   1:  PR[91,3] = PR[90,3] + 56.600;
   1:L PR[91] R[100]mm/sec CNT100;
   1:  PR[91,1] = PR[90,1] + 23.637;
   1:  PR[91,2] = PR[90,2] + -23.851;
   1:  PR[91,3] = PR[90,3] + 56.612;
   1:L PR[91] R[100]mm/sec CNT100;
   1:  PR[91,1] = PR[90,1] + 29.260;
   1:  PR[91,2] = PR[90,2] + -22.769;
   1:  PR[91,3] = PR[90,3] + 56.618;
   1:L PR[91] R[100]mm/sec CNT100;
   1:  PR[91,1] = PR[90,1] + 29.704;
   1:  PR[91,2] = PR[90,2] + -22.625;
   1:  PR[91,3] = PR[90,3] + 56.637;
   1:L PR[91] R[100]mm/sec CNT100;
   1:  PR[91,1] = PR[90,1] + 30.561;
   1:  PR[91,2] = PR[90,2] + -22.294;
   1:  PR[91,3] = PR[90,3] + 56.639;
   1:L PR[91] R[100]mm/sec CNT100;
   1:  PR[91,1] = PR[90,1] + 33.444;
   1:  PR[91,2] = PR[90,2] + -20.954;
   1:  PR[91,3] = PR[90,3] + 56.642;
   1:L PR[91] R[100]mm/sec CNT100;
   1:  PR[91,1] = PR[90,1] + 37.250;
   1:  PR[91,2] = PR[90,2] + -22.447;
   1:  PR[91,3] = PR[90,3] + 56.652;
   1:L PR[91] R[100]mm/sec CNT100;
   1:  PR[91,1] = PR[90,1] + 37.514;
   1:  PR[91,2] = PR[90,2] + -22.529;
   1:  PR[91,3] = PR[90,3] + 56.666;
   1:L PR[91] R[100]mm/sec CNT100;
   1:  PR[91,1] = PR[90,1] + 38.883;
   1:  PR[91,2] = PR[90,2] + -22.892;
   1:  PR[91,3] = PR[90,3] + 56.667;
   1:L PR[91] R[100]mm/sec CNT100;
   1:  PR[91,1] = PR[90,1] + 41.909;
   1:  PR[91,2] = PR[90,2] + -23.658;
   1:  PR[91,3] = PR[90,3] + 56.671;
   1:L PR[91] R[100]mm/sec CNT100;
   1:  PR[91,1] = PR[90,1] + 45.377;
   1:  PR[91,2] = PR[90,2] + -24.220;
   1:  PR[91,3] = PR[90,3] + 56.682;
   1:L PR[91] R[100]mm/sec CNT100;
   1:  PR[91,1] = PR[90,1] + 46.524;
   1:  PR[91,2] = PR[90,2] + -24.421;
   1:  PR[91,3] = PR[90,3] + 56.693;
   1:L PR[91] R[100]mm/sec CNT100;
   1:  PR[91,1] = PR[90,1] + 50.126;
   1:  PR[91,2] = PR[90,2] + -24.627;
   1:  PR[91,3] = PR[90,3] + 56.697;
   1:L PR[91] R[100]mm/sec CNT100;
   1:  PR[91,1] = PR[90,1] + 55.050;
   1:  PR[91,2] = PR[90,2] + -24.652;
   1:  PR[91,3] = PR[90,3] + 56.709;
   1:L PR[91] R[100]mm/sec CNT100;
   1:  PR[91,1] = PR[90,1] + 55.608;
   1:  PR[91,2] = PR[90,2] + -24.620;
   1:  PR[91,3] = PR[90,3] + 56.725;
   1:L PR[91] R[100]mm/sec CNT100;
   1:  PR[91,1] = PR[90,1] + 60.745;
   1:  PR[91,2] = PR[90,2] + -23.797;
   1:  PR[91,3] = PR[90,3] + 56.727;
   1:L PR[91] R[100]mm/sec CNT100;
   1:  PR[91,1] = PR[90,1] + 62.719;
   1:  PR[91,2] = PR[90,2] + -23.452;
   1:  PR[91,3] = PR[90,3] + 56.744;
   1:L PR[91] R[100]mm/sec CNT100;
   1:  PR[91,1] = PR[90,1] + 65.264;
   1:  PR[91,2] = PR[90,2] + -22.556;
   1:  PR[91,3] = PR[90,3] + 56.751;
   1:L PR[91] R[100]mm/sec CNT100;
   1:  PR[91,1] = PR[90,1] + 69.091;
   1:  PR[91,2] = PR[90,2] + -21.163;
   1:  PR[91,3] = PR[90,3] + 56.760;
   1:L PR[91] R[100]mm/sec CNT100;
   1:  PR[91,1] = PR[90,1] + 71.668;
   1:  PR[91,2] = PR[90,2] + -19.643;
   1:  PR[91,3] = PR[90,3] + 56.773;
   1:L PR[91] R[100]mm/sec CNT100;
   1:  PR[91,1] = PR[90,1] + 74.000;
   1:  PR[91,2] = PR[90,2] + -18.185;
   1:  PR[91,3] = PR[90,3] + 56.783;
   1:L PR[91] R[100]mm/sec CNT100;
   1:  PR[91,1] = PR[90,1] + 74.562;
   1:  PR[91,2] = PR[90,2] + -17.699;
   1:  PR[91,3] = PR[90,3] + 56.792;
   1:L PR[91] R[100]mm/sec CNT100;
   1:  PR[91,1] = PR[90,1] + 77.771;
   1:  PR[91,2] = PR[90,2] + -14.617;
   1:  PR[91,3] = PR[90,3] + 56.794;
   1:L PR[91] R[100]mm/sec CNT100;
   1:  PR[91,1] = PR[90,1] + 78.956;
   1:  PR[91,2] = PR[90,2] + -12.985;
   1:  PR[91,3] = PR[90,3] + 56.809;
   1:L PR[91] R[100]mm/sec CNT100;
   1:  PR[91,1] = PR[90,1] + 80.681;
   1:  PR[91,2] = PR[90,2] + -10.394;
   1:  PR[91,3] = PR[90,3] + 56.816;
   1:L PR[91] R[100]mm/sec CNT100;
   1:  PR[91,1] = PR[90,1] + 81.711;
   1:  PR[91,2] = PR[90,2] + -7.850;
   1:  PR[91,3] = PR[90,3] + 56.826;
   1:L PR[91] R[100]mm/sec CNT100;
   1:  PR[91,1] = PR[90,1] + 82.517;
   1:  PR[91,2] = PR[90,2] + -5.690;
   1:  PR[91,3] = PR[90,3] + 56.835;
   1:L PR[91] R[100]mm/sec CNT100;
   1:  PR[91,1] = PR[90,1] + 82.929;
   1:  PR[91,2] = PR[90,2] + -2.575;
   1:  PR[91,3] = PR[90,3] + 56.843;
   1:L PR[91] R[100]mm/sec CNT100;
   1:  PR[91,1] = PR[90,1] + 83.277;
   1:  PR[91,2] = PR[90,2] + -0.677;
   1:  PR[91,3] = PR[90,3] + 56.853;
   1:L PR[91] R[100]mm/sec CNT100;
   1:  PR[91,1] = PR[90,1] + 83.183;
   1:  PR[91,2] = PR[90,2] + 0.041;
   1:  PR[91,3] = PR[90,3] + 56.859;
   1:L PR[91] R[100]mm/sec CNT100;
   1:  PR[91,1] = PR[90,1] + 82.753;
   1:  PR[91,2] = PR[90,2] + 2.220;
   1:  PR[91,3] = PR[90,3] + 56.862;
   1:L PR[91] R[100]mm/sec CNT100;
   1:  PR[91,1] = PR[90,1] + 82.512;
   1:  PR[91,2] = PR[90,2] + 4.246;
   1:  PR[91,3] = PR[90,3] + 56.869;
   1:L PR[91] R[100]mm/sec CNT100;
   1:  PR[91,1] = PR[90,1] + 81.707;
   1:  PR[91,2] = PR[90,2] + 6.399;
   1:  PR[91,3] = PR[90,3] + 56.876;
   1:L PR[91] R[100]mm/sec CNT100;
   1:  PR[91,1] = PR[90,1] + 80.678;
   1:  PR[91,2] = PR[90,2] + 8.942;
   1:  PR[91,3] = PR[90,3] + 56.883;
   1:L PR[91] R[100]mm/sec CNT100;
   1:  PR[91,1] = PR[90,1] + 78.944;
   1:  PR[91,2] = PR[90,2] + 11.541;
   1:  PR[91,3] = PR[90,3] + 56.892;
   1:L PR[91] R[100]mm/sec CNT100;
   1:  PR[91,1] = PR[90,1] + 77.761;
   1:  PR[91,2] = PR[90,2] + 13.171;
   1:  PR[91,3] = PR[90,3] + 56.903;
   1:L PR[91] R[100]mm/sec CNT100;
   1:  PR[91,1] = PR[90,1] + 74.532;
   1:  PR[91,2] = PR[90,2] + 16.264;
   1:  PR[91,3] = PR[90,3] + 56.909;
   1:L PR[91] R[100]mm/sec CNT100;
   1:  PR[91,1] = PR[90,1] + 73.976;
   1:  PR[91,2] = PR[90,2] + 16.745;
   1:  PR[91,3] = PR[90,3] + 56.924;
   1:L PR[91] R[100]mm/sec CNT100;
   1:  PR[91,1] = PR[90,1] + 71.670;
   1:  PR[91,2] = PR[90,2] + 18.183;
   1:  PR[91,3] = PR[90,3] + 56.926;
   1:L PR[91] R[100]mm/sec CNT100;
   1:  PR[91,1] = PR[90,1] + 69.055;
   1:  PR[91,2] = PR[90,2] + 19.721;
   1:  PR[91,3] = PR[90,3] + 56.935;
   1:L PR[91] R[100]mm/sec CNT100;
   1:  PR[91,1] = PR[90,1] + 65.241;
   1:  PR[91,2] = PR[90,2] + 21.101;
   1:  PR[91,3] = PR[90,3] + 56.945;
   1:L PR[91] R[100]mm/sec CNT100;
   1:  PR[91,1] = PR[90,1] + 62.707;
   1:  PR[91,2] = PR[90,2] + 21.996;
   1:  PR[91,3] = PR[90,3] + 56.959;
   1:L PR[91] R[100]mm/sec CNT100;
   1:  PR[91,1] = PR[90,1] + 60.741;
   1:  PR[91,2] = PR[90,2] + 22.335;
   1:  PR[91,3] = PR[90,3] + 56.968;
   1:L PR[91] R[100]mm/sec CNT100;
   1:  PR[91,1] = PR[90,1] + 55.634;
   1:  PR[91,2] = PR[90,2] + 23.160;
   1:  PR[91,3] = PR[90,3] + 56.974;
   1:L PR[91] R[100]mm/sec CNT100;
   1:  PR[91,1] = PR[90,1] + 55.091;
   1:  PR[91,2] = PR[90,2] + 23.191;
   1:  PR[91,3] = PR[90,3] + 56.991;
   1:L PR[91] R[100]mm/sec CNT100;
   1:  PR[91,1] = PR[90,1] + 50.139;
   1:  PR[91,2] = PR[90,2] + 23.170;
   1:  PR[91,3] = PR[90,3] + 56.993;
   1:L PR[91] R[100]mm/sec CNT100;
   1:  PR[91,1] = PR[90,1] + 46.529;
   1:  PR[91,2] = PR[90,2] + 22.962;
   1:  PR[91,3] = PR[90,3] + 57.009;
   1:L PR[91] R[100]mm/sec CNT100;
   1:  PR[91,1] = PR[90,1] + 45.377;
   1:  PR[91,2] = PR[90,2] + 22.761;
   1:  PR[91,3] = PR[90,3] + 57.021;
   1:L PR[91] R[100]mm/sec CNT100;
   1:  PR[91,1] = PR[90,1] + 41.909;
   1:  PR[91,2] = PR[90,2] + 22.199;
   1:  PR[91,3] = PR[90,3] + 57.025;
   1:L PR[91] R[100]mm/sec CNT100;
   1:  PR[91,1] = PR[90,1] + 38.883;
   1:  PR[91,2] = PR[90,2] + 21.434;
   1:  PR[91,3] = PR[90,3] + 57.037;
   1:L PR[91] R[100]mm/sec CNT100;
   1:  PR[91,1] = PR[90,1] + 37.514;
   1:  PR[91,2] = PR[90,2] + 21.070;
   1:  PR[91,3] = PR[90,3] + 57.047;
   1:L PR[91] R[100]mm/sec CNT100;
   1:  PR[91,1] = PR[90,1] + 37.250;
   1:  PR[91,2] = PR[90,2] + 20.988;
   1:  PR[91,3] = PR[90,3] + 57.052;
   1:L PR[91] R[100]mm/sec CNT100;
   1:  PR[91,1] = PR[90,1] + 33.444;
   1:  PR[91,2] = PR[90,2] + 19.495;
   1:  PR[91,3] = PR[90,3] + 57.053;
   1:L PR[91] R[100]mm/sec CNT100;
   1:  PR[91,1] = PR[90,1] + 30.562;
   1:  PR[91,2] = PR[90,2] + 20.835;
   1:  PR[91,3] = PR[90,3] + 57.066;
   1:L PR[91] R[100]mm/sec CNT100;
   1:  PR[91,1] = PR[90,1] + 29.701;
   1:  PR[91,2] = PR[90,2] + 21.168;
   1:  PR[91,3] = PR[90,3] + 57.077;
   1:L PR[91] R[100]mm/sec CNT100;
   1:  PR[91,1] = PR[90,1] + 29.320;
   1:  PR[91,2] = PR[90,2] + 21.293;
   1:  PR[91,3] = PR[90,3] + 57.080;
   1:L PR[91] R[100]mm/sec CNT100;
   1:  PR[91,1] = PR[90,1] + 25.439;
   1:  PR[91,2] = PR[90,2] + 22.057;
   1:  PR[91,3] = PR[90,3] + 57.081;
   1:L PR[91] R[100]mm/sec CNT100;
   1:  PR[91,1] = PR[90,1] + 23.646;
   1:  PR[91,2] = PR[90,2] + 22.392;
   1:  PR[91,3] = PR[90,3] + 57.094;
   1:L PR[91] R[100]mm/sec CNT100;
   1:  PR[91,1] = PR[90,1] + 21.624;
   1:  PR[91,2] = PR[90,2] + 22.312;
   1:  PR[91,3] = PR[90,3] + 57.100;
   1:L PR[91] R[100]mm/sec CNT100;
   1:  PR[91,1] = PR[90,1] + 18.051;
   1:  PR[91,2] = PR[90,2] + 22.116;
   1:  PR[91,3] = PR[90,3] + 57.107;
   1:L PR[91] R[100]mm/sec CNT100;
   1:  PR[91,1] = PR[90,1] + 15.863;
   1:  PR[91,2] = PR[90,2] + 21.519;
   1:  PR[91,3] = PR[90,3] + 57.118;
   1:L PR[91] R[100]mm/sec CNT100;
   1:  PR[91,1] = PR[90,1] + 12.714;
   1:  PR[91,2] = PR[90,2] + 20.535;
   1:  PR[91,3] = PR[90,3] + 57.126;
   1:L PR[91] R[100]mm/sec CNT100;
   1:  PR[91,1] = PR[90,1] + 10.446;
   1:  PR[91,2] = PR[90,2] + 19.306;
   1:  PR[91,3] = PR[90,3] + 57.137;
   1:L PR[91] R[100]mm/sec CNT100;
   1:  PR[91,1] = PR[90,1] + 7.875;
   1:  PR[91,2] = PR[90,2] + 17.717;
   1:  PR[91,3] = PR[90,3] + 57.145;
   1:L PR[91] R[100]mm/sec CNT100;
   1:  PR[91,1] = PR[90,1] + 6.403;
   1:  PR[91,2] = PR[90,2] + 16.502;
   1:  PR[91,3] = PR[90,3] + 57.155;
   1:L PR[91] R[100]mm/sec CNT100;
   1:  PR[91,1] = PR[90,1] + 4.585;
   1:  PR[91,2] = PR[90,2] + 14.804;
   1:  PR[91,3] = PR[90,3] + 57.162;
   1:L PR[91] R[100]mm/sec CNT100;
   1:  PR[91,1] = PR[90,1] + 2.990;
   1:  PR[91,2] = PR[90,2] + 16.205;
   1:  PR[91,3] = PR[90,3] + 57.170;
   1:L PR[91] R[100]mm/sec CNT100;
   1:  PR[91,1] = PR[90,1] + 2.493;
   1:  PR[91,2] = PR[90,2] + 16.511;
   1:  PR[91,3] = PR[90,3] + 57.177;
   1:L PR[91] R[100]mm/sec CNT100;
   1:  PR[91,1] = PR[90,1] + -1.649;
   1:  PR[91,2] = PR[90,2] + 18.902;
   1:  PR[91,3] = PR[90,3] + 57.179;
   1:L PR[91] R[100]mm/sec CNT100;
   1:  PR[91,1] = PR[90,1] + -3.802;
   1:  PR[91,2] = PR[90,2] + 19.647;
   1:  PR[91,3] = PR[90,3] + 57.194;
   1:L PR[91] R[100]mm/sec CNT100;
   1:  PR[91,1] = PR[90,1] + -6.841;
   1:  PR[91,2] = PR[90,2] + 20.634;
   1:  PR[91,3] = PR[90,3] + 57.202;
   1:L PR[91] R[100]mm/sec CNT100;
   1:  PR[91,1] = PR[90,1] + -10.789;
   1:  PR[91,2] = PR[90,2] + 21.127;
   1:  PR[91,3] = PR[90,3] + 57.212;
   1:L PR[91] R[100]mm/sec CNT100;
   1:  PR[91,1] = PR[90,1] + -12.398;
   1:  PR[91,2] = PR[90,2] + 21.314;
   1:  PR[91,3] = PR[90,3] + 57.226;
   1:L PR[91] R[100]mm/sec CNT100;
   1:  PR[91,1] = PR[90,1] + -13.335;
   1:  PR[91,2] = PR[90,2] + 21.242;
   1:  PR[91,3] = PR[90,3] + 57.231;
   1:L PR[91] R[100]mm/sec CNT100;
   1:  PR[91,1] = PR[90,1] + -18.030;
   1:  PR[91,2] = PR[90,2] + 20.872;
   1:  PR[91,3] = PR[90,3] + 57.234;
   1:L PR[91] R[100]mm/sec CNT100;
   1:  PR[91,1] = PR[90,1] + -22.974;
   1:  PR[91,2] = PR[90,2] + 19.453;
   1:  PR[91,3] = PR[90,3] + 57.250;
   1:L PR[91] R[100]mm/sec CNT100;
   1:  PR[91,1] = PR[90,1] + -23.418;
   1:  PR[91,2] = PR[90,2] + 19.263;
   1:  PR[91,3] = PR[90,3] + 57.266;
   1:L PR[91] R[100]mm/sec CNT100;
   1:  PR[91,1] = PR[90,1] + -27.254;
   1:  PR[91,2] = PR[90,2] + 17.207;
   1:  PR[91,3] = PR[90,3] + 57.268;
   1:L PR[91] R[100]mm/sec CNT100;
   1:  PR[91,1] = PR[90,1] + -28.344;
   1:  PR[91,2] = PR[90,2] + 16.438;
   1:  PR[91,3] = PR[90,3] + 57.282;
   1:L PR[91] R[100]mm/sec CNT100;
   1:  PR[91,1] = PR[90,1] + -28.555;
   1:  PR[91,2] = PR[90,2] + 16.310;
   1:  PR[91,3] = PR[90,3] + 57.287;
   1:L PR[91] R[100]mm/sec CNT100;
   1:  PR[91,1] = PR[90,1] + -30.574;
   1:  PR[91,2] = PR[90,2] + 14.844;
   1:  PR[91,3] = PR[90,3] + 57.288;
   1:L PR[91] R[100]mm/sec CNT100;
   1:  PR[91,1] = PR[90,1] + -35.677;
   1:  PR[91,2] = PR[90,2] + 16.912;
   1:  PR[91,3] = PR[90,3] + 57.296;
   1:L PR[91] R[100]mm/sec CNT100;
   1:  PR[91,1] = PR[90,1] + -36.847;
   1:  PR[91,2] = PR[90,2] + 17.527;
   1:  PR[91,3] = PR[90,3] + 57.314;
   1:L PR[91] R[100]mm/sec CNT100;
   1:  PR[91,1] = PR[90,1] + -37.867;
   1:  PR[91,2] = PR[90,2] + 17.950;
   1:  PR[91,3] = PR[90,3] + 57.318;
   1:L PR[91] R[100]mm/sec CNT100;
   1:  PR[91,1] = PR[90,1] + -41.482;
   1:  PR[91,2] = PR[90,2] + 19.050;
   1:  PR[91,3] = PR[90,3] + 57.322;
   1:L PR[91] R[100]mm/sec CNT100;
   1:  PR[91,1] = PR[90,1] + -45.232;
   1:  PR[91,2] = PR[90,2] + 19.915;
   1:  PR[91,3] = PR[90,3] + 57.334;
   1:L PR[91] R[100]mm/sec CNT100;
   1:  PR[91,1] = PR[90,1] + -47.004;
   1:  PR[91,2] = PR[90,2] + 20.403;
   1:  PR[91,3] = PR[90,3] + 57.347;
   1:L PR[91] R[100]mm/sec CNT100;
   1:  PR[91,1] = PR[90,1] + -50.693;
   1:  PR[91,2] = PR[90,2] + 20.804;
   1:  PR[91,3] = PR[90,3] + 57.353;
   1:L PR[91] R[100]mm/sec CNT100;
   1:  PR[91,1] = PR[90,1] + -54.131;
   1:  PR[91,2] = PR[90,2] + 21.124;
   1:  PR[91,3] = PR[90,3] + 57.365;
   1:L PR[91] R[100]mm/sec CNT100;
   1:  PR[91,1] = PR[90,1] + -59.648;
   1:  PR[91,2] = PR[90,2] + 20.809;
   1:  PR[91,3] = PR[90,3] + 57.377;
   1:L PR[91] R[100]mm/sec CNT100;
   1:  PR[91] = PR[90];
   1:  PR[91,1] = PR[90,1] + -63.521;
   1:  PR[91,2] = PR[90,2] + 20.021;
   1:  PR[91,3] = PR[90,3] + 58.695;
   1:L PR[91] R[100]mm/sec CNT100;
   1:  PR[91,1] = PR[90,1] + -65.346;
   1:  PR[91,2] = PR[90,2] + 19.577;
   1:  PR[91,3] = PR[90,3] + 57.408;
   1:L PR[91] R[100]mm/sec CNT100;
   1:  PR[91,1] = PR[90,1] + -67.455;
   1:  PR[91,2] = PR[90,2] + 18.685;
   1:  PR[91,3] = PR[90,3] + 57.415;
   1:L PR[91] R[100]mm/sec CNT100;
   1:  PR[91,1] = PR[90,1] + -70.428;
   1:  PR[91,2] = PR[90,2] + 17.390;
   1:  PR[91,3] = PR[90,3] + 57.422;
   1:L PR[91] R[100]mm/sec CNT100;
   1:  PR[91,1] = PR[90,1] + -74.679;
   1:  PR[91,2] = PR[90,2] + 14.541;
   1:  PR[91,3] = PR[90,3] + 57.433;
   1:L PR[91] R[100]mm/sec CNT100;
   1:  PR[91,1] = PR[90,1] + -77.809;
   1:  PR[91,2] = PR[90,2] + 11.230;
   1:  PR[91,3] = PR[90,3] + 57.450;
   1:L PR[91] R[100]mm/sec CNT100;
   1:  PR[91,1] = PR[90,1] + -80.119;
   1:  PR[91,2] = PR[90,2] + 7.477;
   1:  PR[91,3] = PR[90,3] + 57.465;
   1:L PR[91] R[100]mm/sec CNT100;
   1:  PR[91,1] = PR[90,1] + -81.526;
   1:  PR[91,2] = PR[90,2] + 3.442;
   1:  PR[91,3] = PR[90,3] + 57.480;
   1:L PR[91] R[100]mm/sec CNT100;
   1:  PR[91,1] = PR[90,1] + -81.701;
   1:  PR[91,2] = PR[90,2] + 1.923;
   1:  PR[91,3] = PR[90,3] + 57.494;
   1:L PR[91] R[100]mm/sec CNT100;
   1:  PR[91,1] = PR[90,1] + -81.979;
   1:  PR[91,2] = PR[90,2] + 0.421;
   1:  PR[91,3] = PR[90,3] + 57.499;
   1:L PR[91] R[100]mm/sec CNT100;
   1:  PR[91,1] = PR[90,1] + -82.105;
   1:  PR[91,2] = PR[90,2] + -0.448;
   1:  PR[91,3] = PR[90,3] + 57.505;
   1:L PR[91] R[100]mm/sec CNT100;
   1:  PR[91,1] = PR[90,1] + -82.136;
   1:  PR[91,2] = PR[90,2] + -0.719;
   1:  PR[91,3] = PR[90,3] + 57.508;
   1:L PR[91] R[100]mm/sec CNT100;
   1:  PR[91,1] = PR[90,1] + -81.791;
   1:  PR[91,2] = PR[90,2] + -3.476;
   1:L PR[91] R[100]mm/sec CNT100;
   1:  PR[91,1] = PR[90,1] + -81.638;
   1:  PR[91,2] = PR[90,2] + -4.207;
   1:  PR[91,3] = PR[90,3] + 57.518;
   1:L PR[91] R[100]mm/sec CNT100;
   1:  PR[91,1] = PR[90,1] + -81.550;
   1:  PR[91,2] = PR[90,2] + -4.931;
   1:  PR[91,3] = PR[90,3] + 57.520;
   1:L PR[91] R[100]mm/sec CNT100;
   1:  PR[91,1] = PR[90,1] + -80.396;
   1:  PR[91,2] = PR[90,2] + -8.144;
   1:  PR[91,3] = PR[90,3] + 57.523;
   1:L PR[91] R[100]mm/sec CNT100;
   1:  PR[91,1] = PR[90,1] + -80.063;
   1:  PR[91,2] = PR[90,2] + -9.024;
   1:  PR[91,3] = PR[90,3] + 57.534;
   1:L PR[91] R[100]mm/sec CNT100;
   1:  PR[91,1] = PR[90,1] + -78.391;
   1:  PR[91,2] = PR[90,2] + -11.659;
   1:  PR[91,3] = PR[90,3] + 57.537;
   1:L PR[91] R[100]mm/sec CNT100;
   1:  PR[91,1] = PR[90,1] + -77.560;
   1:  PR[91,2] = PR[90,2] + -12.896;
   1:  PR[91,3] = PR[90,3] + 57.548;
   1:L PR[91] R[100]mm/sec CNT100;
   1:  PR[91,1] = PR[90,1] + -75.708;
   1:  PR[91,2] = PR[90,2] + -14.796;
   1:  PR[91,3] = PR[90,3] + 57.553;
   1:L PR[91] R[100]mm/sec CNT100;
   1:  PR[91,1] = PR[90,1] + -74.027;
   1:  PR[91,2] = PR[90,2] + -16.398;
   1:  PR[91,3] = PR[90,3] + 57.561;
   1:L PR[91] R[100]mm/sec CNT100;
   1:  PR[91,1] = PR[90,1] + -72.425;
   1:  PR[91,2] = PR[90,2] + -17.499;
   1:  PR[91,3] = PR[90,3] + 57.569;
   1:L PR[91] R[100]mm/sec CNT100;
   1:  PR[91,1] = PR[90,1] + -69.453;
   1:  PR[91,2] = PR[90,2] + -19.351;
   1:  PR[91,3] = PR[90,3] + 57.576;
   1:L PR[91] R[100]mm/sec CNT100;
   1:  PR[91,1] = PR[90,1] + -68.619;
   1:  PR[91,2] = PR[90,2] + -19.721;
   1:  PR[91,3] = PR[90,3] + 57.587;
   1:L PR[91] R[100]mm/sec CNT100;
   1:  PR[91,1] = PR[90,1] + -65.053;
   1:  PR[91,2] = PR[90,2] + -21.075;
   1:  PR[91,3] = PR[90,3] + 57.590;
   1:L PR[91] R[100]mm/sec CNT100;
   1:  PR[91,1] = PR[90,1] + -63.958;
   1:  PR[91,2] = PR[90,2] + -21.475;
   1:  PR[91,3] = PR[90,3] + 57.603;
   1:L PR[91] R[100]mm/sec CNT100;
   1:  PR[91,1] = PR[90,1] + -57.805;
   1:  PR[91,2] = PR[90,2] + -22.597;
   1:  PR[91,3] = PR[90,3] + 57.607;
   1:L PR[91] R[100]mm/sec CNT100;
   1:  PR[91,1] = PR[90,1] + -51.350;
   1:  PR[91,2] = PR[90,2] + -22.721;
   1:  PR[91,3] = PR[90,3] + 57.628;
   1:L PR[91] R[100]mm/sec CNT100;
   1:  PR[91,1] = PR[90,1] + -50.235;
   1:  PR[91,2] = PR[90,2] + -22.555;
   1:  PR[91,3] = PR[90,3] + 57.649;
   1:L PR[91] R[100]mm/sec CNT100;
   1:  PR[91,1] = PR[90,1] + -45.501;
   1:  PR[91,2] = PR[90,2] + -22.036;
   1:  PR[91,3] = PR[90,3] + 57.653;
   1:L PR[91] R[100]mm/sec CNT100;
   1:  PR[91,1] = PR[90,1] + -41.965;
   1:  PR[91,2] = PR[90,2] + -21.358;
   1:  PR[91,3] = PR[90,3] + 57.669;
   1:L PR[91] R[100]mm/sec CNT100;
   1:  PR[91,1] = PR[90,1] + -40.439;
   1:  PR[91,2] = PR[90,2] + -20.935;
   1:  PR[91,3] = PR[90,3] + 57.681;
   1:L PR[91] R[100]mm/sec CNT100;
   1:  PR[91,1] = PR[90,1] + -38.575;
   1:  PR[91,2] = PR[90,2] + -20.262;
   1:  PR[91,3] = PR[90,3] + 57.686;
   1:L PR[91] R[100]mm/sec CNT100;
   1:  PR[91,1] = PR[90,1] + -35.328;
   1:  PR[91,2] = PR[90,2] + -19.343;
   1:  PR[91,3] = PR[90,3] + 57.693;
   1:L PR[91] R[100]mm/sec CNT100;
   1:  PR[91,1] = PR[90,1] + -31.914;
   1:  PR[91,2] = PR[90,2] + -18.110;
   1:  PR[91,3] = PR[90,3] + 57.704;
   1:L PR[91] R[100]mm/sec CNT100;
   1:  PR[91,1] = PR[90,1] + -29.374;
   1:  PR[91,2] = PR[90,2] + -16.925;
   1:  PR[91,3] = PR[90,3] + 57.716;
   1:L PR[91] R[100]mm/sec CNT100;
   1:  PR[91,1] = PR[90,1] + -28.132;
   1:  PR[91,2] = PR[90,2] + -17.957;
   1:  PR[91,3] = PR[90,3] + 57.726;
   1:L PR[91] R[100]mm/sec CNT100;
   1:  PR[91,1] = PR[90,1] + -27.145;
   1:  PR[91,2] = PR[90,2] + -18.622;
   1:  PR[91,3] = PR[90,3] + 57.731;
   1:L PR[91] R[100]mm/sec CNT100;
   1:  PR[91,1] = PR[90,1] + -22.761;
   1:  PR[91,2] = PR[90,2] + -20.984;
   1:  PR[91,3] = PR[90,3] + 57.735;
   1:L PR[91] R[100]mm/sec CNT100;
   1:  PR[91,1] = PR[90,1] + -17.923;
   1:  PR[91,2] = PR[90,2] + -22.392;
   1:  PR[91,3] = PR[90,3] + 57.751;
   1:L PR[91] R[100]mm/sec CNT100;
   1:  PR[91,1] = PR[90,1] + -17.426;
   1:  PR[91,2] = PR[90,2] + -22.525;
   1:  PR[91,3] = PR[90,3] + 57.768;
   1:L PR[91] R[100]mm/sec CNT100;
   1:  PR[91,1] = PR[90,1] + -11.769;
   1:  PR[91,2] = PR[90,2] + -22.973;
   1:  PR[91,3] = PR[90,3] + 57.770;
   1:L PR[91] R[100]mm/sec CNT100;
   1:  PR[91,1] = PR[90,1] + -8.735;
   1:  PR[91,2] = PR[90,2] + -22.592;
   1:  PR[91,3] = PR[90,3] + 57.789;
   1:L PR[91] R[100]mm/sec CNT100;
   1:  PR[91,1] = PR[90,1] + -6.180;
   1:  PR[91,2] = PR[90,2] + -22.303;
   1:  PR[91,3] = PR[90,3] + 57.799;
   1:L PR[91] R[100]mm/sec CNT100;
   1:  PR[91,1] = PR[90,1] + -2.208;
   1:  PR[91,2] = PR[90,2] + -21.016;
   1:  PR[91,3] = PR[90,3] + 57.808;
   1:L PR[91] R[100]mm/sec CNT100;
   1:  PR[91,1] = PR[90,1] + -0.980;
   1:  PR[91,2] = PR[90,2] + -20.593;
   1:  PR[91,3] = PR[90,3] + 57.822;
   1:L PR[91] R[100]mm/sec CNT100;
   1:  PR[91,1] = PR[90,1] + 3.412;
   1:  PR[91,2] = PR[90,2] + -18.069;
   1:  PR[91,3] = PR[90,3] + 57.826;
   1:L PR[91] R[100]mm/sec CNT100;
   1:  PR[91,1] = PR[90,1] + 5.084;
   1:  PR[91,2] = PR[90,2] + -17.207;
   1:  PR[91,3] = PR[90,3] + 57.843;
   1:L PR[91] R[100]mm/sec CNT100;
   1:  PR[91,1] = PR[90,1] + 6.725;
   1:  PR[91,2] = PR[90,2] + -18.651;
   1:  PR[91,3] = PR[90,3] + 57.849;
   1:L PR[91] R[100]mm/sec CNT100;
   1:  PR[91,1] = PR[90,1] + 7.716;
   1:  PR[91,2] = PR[90,2] + -19.429;
   1:  PR[91,3] = PR[90,3] + 57.856;
   1:L PR[91] R[100]mm/sec CNT100;
   1:  PR[91,1] = PR[90,1] + 9.813;
   1:  PR[91,2] = PR[90,2] + -20.725;
   1:  PR[91,3] = PR[90,3] + 57.861;
   1:L PR[91] R[100]mm/sec CNT100;
   1:  PR[91,1] = PR[90,1] + 12.586;
   1:  PR[91,2] = PR[90,2] + -22.227;
   1:  PR[91,3] = PR[90,3] + 57.869;
   1:L PR[91] R[100]mm/sec CNT100;
   1:  PR[91,1] = PR[90,1] + 15.184;
   1:  PR[91,2] = PR[90,2] + -23.040;
   1:  PR[91,3] = PR[90,3] + 57.879;
   1:L PR[91] R[100]mm/sec CNT100;
   1:  PR[91,1] = PR[90,1] + 17.927;
   1:  PR[91,2] = PR[90,2] + -23.788;
   1:  PR[91,3] = PR[90,3] + 57.888;
   1:L PR[91] R[100]mm/sec CNT100;
   1:  PR[91,1] = PR[90,1] + 20.928;
   1:  PR[91,2] = PR[90,2] + -23.953;
   1:  PR[91,3] = PR[90,3] + 57.898;
   1:L PR[91] R[100]mm/sec CNT100;
   1:  PR[91,1] = PR[90,1] + 23.513;
   1:  PR[91,2] = PR[90,2] + -24.056;
   1:  PR[91,3] = PR[90,3] + 57.908;
   1:L PR[91] R[100]mm/sec CNT100;
   1:  PR[91,1] = PR[90,1] + 26.736;
   1:  PR[91,2] = PR[90,2] + -23.428;
   1:  PR[91,3] = PR[90,3] + 57.917;
   1:L PR[91] R[100]mm/sec CNT100;
   1:  PR[91,1] = PR[90,1] + 29.137;
   1:  PR[91,2] = PR[90,2] + -22.977;
   1:  PR[91,3] = PR[90,3] + 57.928;
   1:L PR[91] R[100]mm/sec CNT100;
   1:  PR[91,1] = PR[90,1] + 29.749;
   1:  PR[91,2] = PR[90,2] + -22.780;
   1:  PR[91,3] = PR[90,3] + 57.936;
   1:L PR[91] R[100]mm/sec CNT100;
   1:  PR[91,1] = PR[90,1] + 30.881;
   1:  PR[91,2] = PR[90,2] + -22.342;
   1:  PR[91,3] = PR[90,3] + 57.938;
   1:L PR[91] R[100]mm/sec CNT100;
   1:  PR[91,1] = PR[90,1] + 32.767;
   1:  PR[91,2] = PR[90,2] + -21.466;
   1:  PR[91,3] = PR[90,3] + 57.942;
   1:L PR[91] R[100]mm/sec CNT100;
   1:  PR[91,1] = PR[90,1] + 35.157;
   1:  PR[91,2] = PR[90,2] + -22.403;
   1:  PR[91,3] = PR[90,3] + 57.949;
   1:L PR[91] R[100]mm/sec CNT100;
   1:  PR[91,1] = PR[90,1] + 36.106;
   1:  PR[91,2] = PR[90,2] + -22.696;
   1:  PR[91,3] = PR[90,3] + 57.957;
   1:L PR[91] R[100]mm/sec CNT100;
   1:  PR[91,1] = PR[90,1] + 40.078;
   1:  PR[91,2] = PR[90,2] + -23.752;
   1:  PR[91,3] = PR[90,3] + 57.961;
   1:L PR[91] R[100]mm/sec CNT100;
   1:  PR[91,1] = PR[90,1] + 41.285;
   1:  PR[91,2] = PR[90,2] + -24.057;
   1:  PR[91,3] = PR[90,3] + 57.974;
   1:L PR[91] R[100]mm/sec CNT100;
   1:  PR[91,1] = PR[90,1] + 43.631;
   1:  PR[91,2] = PR[90,2] + -24.437;
   1:  PR[91,3] = PR[90,3] + 57.979;
   1:L PR[91] R[100]mm/sec CNT100;
   1:  PR[91,1] = PR[90,1] + 45.413;
   1:  PR[91,2] = PR[90,2] + -24.670;
   1:  PR[91,3] = PR[90,3] + 57.986;
   1:L PR[91] R[100]mm/sec CNT100;
   1:  PR[91,1] = PR[90,1] + 46.340;
   1:  PR[91,2] = PR[90,2] + -24.709;
   1:  PR[91,3] = PR[90,3] + 57.992;
   1:L PR[91] R[100]mm/sec CNT100;
   1:  PR[91,1] = PR[90,1] + 49.633;
   1:  PR[91,2] = PR[90,2] + -24.898;
   1:  PR[91,3] = PR[90,3] + 57.996;
   1:L PR[91] R[100]mm/sec CNT100;
   1:  PR[91,1] = PR[90,1] + 52.860;
   1:  PR[91,2] = PR[90,2] + -24.915;
   1:  PR[91,3] = PR[90,3] + 58.007;
   1:L PR[91] R[100]mm/sec CNT100;
   1:  PR[91,1] = PR[90,1] + 54.860;
   1:  PR[91,2] = PR[90,2] + -24.798;
   1:  PR[91,3] = PR[90,3] + 58.017;
   1:L PR[91] R[100]mm/sec CNT100;
   1:  PR[91,1] = PR[90,1] + 60.575;
   1:  PR[91,2] = PR[90,2] + -23.888;
   1:  PR[91,3] = PR[90,3] + 58.024;
   1:L PR[91] R[100]mm/sec CNT100;
   1:  PR[91,1] = PR[90,1] + 61.668;
   1:  PR[91,2] = PR[90,2] + -23.697;
   1:  PR[91,3] = PR[90,3] + 58.043;
   1:L PR[91] R[100]mm/sec CNT100;
   1:  PR[91,1] = PR[90,1] + 65.065;
   1:  PR[91,2] = PR[90,2] + -22.501;
   1:  PR[91,3] = PR[90,3] + 58.047;
   1:L PR[91] R[100]mm/sec CNT100;
   1:  PR[91,1] = PR[90,1] + 68.135;
   1:  PR[91,2] = PR[90,2] + -21.384;
   1:  PR[91,3] = PR[90,3] + 58.059;
   1:L PR[91] R[100]mm/sec CNT100;
   1:  PR[91,1] = PR[90,1] + 69.368;
   1:  PR[91,2] = PR[90,2] + -20.667;
   1:  PR[91,3] = PR[90,3] + 58.070;
   1:L PR[91] R[100]mm/sec CNT100;
   1:  PR[91,1] = PR[90,1] + 73.500;
   1:  PR[91,2] = PR[90,2] + -18.216;
   1:  PR[91,3] = PR[90,3] + 58.075;
   1:L PR[91] R[100]mm/sec CNT100;
   1:  PR[91,1] = PR[90,1] + 77.253;
   1:  PR[91,2] = PR[90,2] + -14.615;
   1:  PR[91,3] = PR[90,3] + 58.091;
   1:L PR[91] R[100]mm/sec CNT100;
   1:  PR[91,1] = PR[90,1] + 77.951;
   1:  PR[91,2] = PR[90,2] + -13.654;
   1:  PR[91,3] = PR[90,3] + 58.108;
   1:L PR[91] R[100]mm/sec CNT100;
   1:  PR[91,1] = PR[90,1] + 80.128;
   1:  PR[91,2] = PR[90,2] + -10.384;
   1:  PR[91,3] = PR[90,3] + 58.112;
   1:L PR[91] R[100]mm/sec CNT100;
   1:  PR[91,1] = PR[90,1] + 80.874;
   1:  PR[91,2] = PR[90,2] + -8.540;
   1:  PR[91,3] = PR[90,3] + 58.125;
   1:L PR[91] R[100]mm/sec CNT100;
   1:  PR[91,1] = PR[90,1] + 81.941;
   1:  PR[91,2] = PR[90,2] + -5.682;
   1:  PR[91,3] = PR[90,3] + 58.132;
   1:L PR[91] R[100]mm/sec CNT100;
   1:  PR[91,1] = PR[90,1] + 82.260;
   1:  PR[91,2] = PR[90,2] + -3.266;
   1:  PR[91,3] = PR[90,3] + 58.142;
   1:L PR[91] R[100]mm/sec CNT100;
   1:  PR[91,1] = PR[90,1] + 82.717;
   1:  PR[91,2] = PR[90,2] + -0.775;
   1:  PR[91,3] = PR[90,3] + 58.150;
   1:L PR[91] R[100]mm/sec CNT100;
   1:  PR[91,1] = PR[90,1] + 82.252;
   1:  PR[91,2] = PR[90,2] + 1.577;
   1:  PR[91,3] = PR[90,3] + 58.158;
   1:L PR[91] R[100]mm/sec CNT100;
   1:  PR[91,1] = PR[90,1] + 81.935;
   1:  PR[91,2] = PR[90,2] + 4.240;
   1:  PR[91,3] = PR[90,3] + 58.166;
   1:L PR[91] R[100]mm/sec CNT100;
   1:  PR[91,1] = PR[90,1] + 80.868;
   1:  PR[91,2] = PR[90,2] + 7.091;
   1:  PR[91,3] = PR[90,3] + 58.175;
   1:L PR[91] R[100]mm/sec CNT100;
   1:  PR[91,1] = PR[90,1] + 80.123;
   1:  PR[91,2] = PR[90,2] + 8.935;
   1:  PR[91,3] = PR[90,3] + 58.186;
   1:L PR[91] R[100]mm/sec CNT100;
   1:  PR[91,1] = PR[90,1] + 77.935;
   1:  PR[91,2] = PR[90,2] + 12.214;
   1:  PR[91,3] = PR[90,3] + 58.192;
   1:L PR[91] R[100]mm/sec CNT100;
   1:  PR[91,1] = PR[90,1] + 77.240;
   1:  PR[91,2] = PR[90,2] + 13.171;
   1:  PR[91,3] = PR[90,3] + 58.205;
   1:L PR[91] R[100]mm/sec CNT100;
   1:  PR[91,1] = PR[90,1] + 73.474;
   1:  PR[91,2] = PR[90,2] + 16.778;
   1:  PR[91,3] = PR[90,3] + 58.209;
   1:L PR[91] R[100]mm/sec CNT100;
   1:  PR[91,1] = PR[90,1] + 69.342;
   1:  PR[91,2] = PR[90,2] + 19.219;
   1:  PR[91,3] = PR[90,3] + 58.227;
   1:L PR[91] R[100]mm/sec CNT100;
   1:  PR[91,1] = PR[90,1] + 68.108;
   1:  PR[91,2] = PR[90,2] + 19.937;
   1:  PR[91,3] = PR[90,3] + 58.243;
   1:L PR[91] R[100]mm/sec CNT100;
   1:  PR[91,1] = PR[90,1] + 65.049;
   1:  PR[91,2] = PR[90,2] + 21.044;
   1:  PR[91,3] = PR[90,3] + 58.247;
   1:L PR[91] R[100]mm/sec CNT100;
   1:  PR[91,1] = PR[90,1] + 61.673;
   1:  PR[91,2] = PR[90,2] + 22.236;
   1:  PR[91,3] = PR[90,3] + 58.258;
   1:L PR[91] R[100]mm/sec CNT100;
   1:  PR[91,1] = PR[90,1] + 60.580;
   1:  PR[91,2] = PR[90,2] + 22.425;
   1:  PR[91,3] = PR[90,3] + 58.270;
   1:L PR[91] R[100]mm/sec CNT100;
   1:  PR[91,1] = PR[90,1] + 54.882;
   1:  PR[91,2] = PR[90,2] + 23.338;
   1:  PR[91,3] = PR[90,3] + 58.274;
   1:L PR[91] R[100]mm/sec CNT100;
   1:  PR[91,1] = PR[90,1] + 52.887;
   1:  PR[91,2] = PR[90,2] + 23.454;
   1:  PR[91,3] = PR[90,3] + 58.293;
   1:L PR[91] R[100]mm/sec CNT100;
   1:  PR[91,1] = PR[90,1] + 49.641;
   1:  PR[91,2] = PR[90,2] + 23.440;
   1:  PR[91,3] = PR[90,3] + 58.300;
   1:L PR[91] R[100]mm/sec CNT100;
   1:  PR[91,1] = PR[90,1] + 46.340;
   1:  PR[91,2] = PR[90,2] + 23.250;
   1:  PR[91,3] = PR[90,3] + 58.311;
   1:L PR[91] R[100]mm/sec CNT100;
   1:  PR[91,1] = PR[90,1] + 45.413;
   1:  PR[91,2] = PR[90,2] + 23.211;
   1:  PR[91,3] = PR[90,3] + 58.322;
   1:L PR[91] R[100]mm/sec CNT100;
   1:  PR[91,1] = PR[90,1] + 43.631;
   1:  PR[91,2] = PR[90,2] + 22.979;
   1:  PR[91,3] = PR[90,3] + 58.325;
   1:L PR[91] R[100]mm/sec CNT100;
   1:  PR[91,1] = PR[90,1] + 41.285;
   1:  PR[91,2] = PR[90,2] + 22.598;
   1:  PR[91,3] = PR[90,3] + 58.331;
   1:L PR[91] R[100]mm/sec CNT100;
   1:  PR[91,1] = PR[90,1] + 40.078;
   1:  PR[91,2] = PR[90,2] + 22.293;
   1:  PR[91,3] = PR[90,3] + 58.339;
   1:L PR[91] R[100]mm/sec CNT100;
   1:  PR[91,1] = PR[90,1] + 36.106;
   1:  PR[91,2] = PR[90,2] + 21.237;
   1:  PR[91,3] = PR[90,3] + 58.343;
   1:L PR[91] R[100]mm/sec CNT100;
   1:  PR[91,1] = PR[90,1] + 35.157;
   1:  PR[91,2] = PR[90,2] + 20.944;
   1:  PR[91,3] = PR[90,3] + 58.357;
   1:L PR[91] R[100]mm/sec CNT100;
   1:  PR[91,1] = PR[90,1] + 32.767;
   1:  PR[91,2] = PR[90,2] + 20.007;
   1:  PR[91,3] = PR[90,3] + 58.360;
   1:L PR[91] R[100]mm/sec CNT100;
   1:  PR[91,1] = PR[90,1] + 30.881;
   1:  PR[91,2] = PR[90,2] + 20.883;
   1:  PR[91,3] = PR[90,3] + 58.368;
   1:L PR[91] R[100]mm/sec CNT100;
   1:  PR[91,1] = PR[90,1] + 29.747;
   1:  PR[91,2] = PR[90,2] + 21.322;
   1:  PR[91,3] = PR[90,3] + 58.375;
   1:L PR[91] R[100]mm/sec CNT100;
   1:  PR[91,1] = PR[90,1] + 29.210;
   1:  PR[91,2] = PR[90,2] + 21.498;
   1:  PR[91,3] = PR[90,3] + 58.379;
   1:L PR[91] R[100]mm/sec CNT100;
   1:  PR[91,1] = PR[90,1] + 25.827;
   1:  PR[91,2] = PR[90,2] + 22.166;
   1:  PR[91,3] = PR[90,3] + 58.381;
   1:L PR[91] R[100]mm/sec CNT100;
   1:  PR[91,1] = PR[90,1] + 23.523;
   1:  PR[91,2] = PR[90,2] + 22.598;
   1:  PR[91,3] = PR[90,3] + 58.393;
   1:L PR[91] R[100]mm/sec CNT100;
   1:  PR[91,1] = PR[90,1] + 20.930;
   1:  PR[91,2] = PR[90,2] + 22.494;
   1:  PR[91,3] = PR[90,3] + 58.401;
   1:L PR[91] R[100]mm/sec CNT100;
   1:  PR[91,1] = PR[90,1] + 17.930;
   1:  PR[91,2] = PR[90,2] + 22.329;
   1:  PR[91,3] = PR[90,3] + 58.409;
   1:L PR[91] R[100]mm/sec CNT100;
   1:  PR[91,1] = PR[90,1] + 15.187;
   1:  PR[91,2] = PR[90,2] + 21.581;
   1:  PR[91,3] = PR[90,3] + 58.419;
   1:L PR[91] R[100]mm/sec CNT100;
   1:  PR[91,1] = PR[90,1] + 12.590;
   1:  PR[91,2] = PR[90,2] + 20.770;
   1:  PR[91,3] = PR[90,3] + 58.429;
   1:L PR[91] R[100]mm/sec CNT100;
   1:  PR[91,1] = PR[90,1] + 9.800;
   1:  PR[91,2] = PR[90,2] + 19.257;
   1:  PR[91,3] = PR[90,3] + 58.438;
   1:L PR[91] R[100]mm/sec CNT100;
   1:  PR[91,1] = PR[90,1] + 7.733;
   1:  PR[91,2] = PR[90,2] + 17.981;
   1:  PR[91,3] = PR[90,3] + 58.448;
   1:L PR[91] R[100]mm/sec CNT100;
   1:  PR[91,1] = PR[90,1] + 5.037;
   1:  PR[91,2] = PR[90,2] + 15.754;
   1:  PR[91,3] = PR[90,3] + 58.456;
   1:L PR[91] R[100]mm/sec CNT100;
   1:  PR[91,1] = PR[90,1] + 3.258;
   1:  PR[91,2] = PR[90,2] + 16.689;
   1:  PR[91,3] = PR[90,3] + 58.468;
   1:L PR[91] R[100]mm/sec CNT100;
   1:  PR[91,1] = PR[90,1] + -0.963;
   1:  PR[91,2] = PR[90,2] + 19.126;
   1:  PR[91,3] = PR[90,3] + 58.475;
   1:L PR[91] R[100]mm/sec CNT100;
   1:  PR[91,1] = PR[90,1] + -2.181;
   1:  PR[91,2] = PR[90,2] + 19.548;
   1:  PR[91,3] = PR[90,3] + 58.491;
   1:L PR[91] R[100]mm/sec CNT100;
   1:  PR[91,1] = PR[90,1] + -6.167;
   1:  PR[91,2] = PR[90,2] + 20.842;
   1:  PR[91,3] = PR[90,3] + 58.495;
   1:L PR[91] R[100]mm/sec CNT100;
   1:  PR[91,1] = PR[90,1] + -9.155;
   1:  PR[91,2] = PR[90,2] + 21.215;
   1:  PR[91,3] = PR[90,3] + 58.509;
   1:L PR[91] R[100]mm/sec CNT100;
   1:  PR[91,1] = PR[90,1] + -11.731;
   1:  PR[91,2] = PR[90,2] + 21.514;
   1:  PR[91,3] = PR[90,3] + 58.519;
   1:L PR[91] R[100]mm/sec CNT100;
   1:  PR[91,1] = PR[90,1] + -17.391;
   1:  PR[91,2] = PR[90,2] + 21.072;
   1:  PR[91,3] = PR[90,3] + 58.528;
   1:L PR[91] R[100]mm/sec CNT100;
   1:  PR[91,1] = PR[90,1] + -17.893;
   1:  PR[91,2] = PR[90,2] + 20.938;
   1:  PR[91,3] = PR[90,3] + 58.547;
   1:L PR[91] R[100]mm/sec CNT100;
   1:  PR[91,1] = PR[90,1] + -22.725;
   1:  PR[91,2] = PR[90,2] + 19.540;
   1:  PR[91,3] = PR[90,3] + 58.549;
   1:L PR[91] R[100]mm/sec CNT100;
   1:  PR[91,1] = PR[90,1] + -27.048;
   1:  PR[91,2] = PR[90,2] + 17.223;
   1:  PR[91,3] = PR[90,3] + 58.566;
   1:L PR[91] R[100]mm/sec CNT100;
   1:  PR[91,1] = PR[90,1] + -27.706;
   1:  PR[91,2] = PR[90,2] + 16.758;
   1:  PR[91,3] = PR[90,3] + 58.582;
   1:L PR[91] R[100]mm/sec CNT100;
   1:  PR[91,1] = PR[90,1] + -27.950;
   1:  PR[91,2] = PR[90,2] + 16.610;
   1:  PR[91,3] = PR[90,3] + 58.585;
   1:L PR[91] R[100]mm/sec CNT100;
   1:  PR[91,1] = PR[90,1] + -29.412;
   1:  PR[91,2] = PR[90,2] + 15.550;
   1:L PR[91] R[100]mm/sec CNT100;
   1:  PR[91,1] = PR[90,1] + -34.506;
   1:  PR[91,2] = PR[90,2] + 17.619;
   1:  PR[91,3] = PR[90,3] + 58.592;
   1:L PR[91] R[100]mm/sec CNT100;
   1:  PR[91,1] = PR[90,1] + -35.673;
   1:  PR[91,2] = PR[90,2] + 18.024;
   1:  PR[91,3] = PR[90,3] + 58.610;
   1:L PR[91] R[100]mm/sec CNT100;
   1:  PR[91,1] = PR[90,1] + -36.381;
   1:  PR[91,2] = PR[90,2] + 18.185;
   1:  PR[91,3] = PR[90,3] + 58.614;
   1:L PR[91] R[100]mm/sec CNT100;
   1:  PR[91,1] = PR[90,1] + -40.836;
   1:  PR[91,2] = PR[90,2] + 19.540;
   1:  PR[91,3] = PR[90,3] + 58.616;
   1:L PR[91] R[100]mm/sec CNT100;
   1:  PR[91,1] = PR[90,1] + -45.220;
   1:  PR[91,2] = PR[90,2] + 20.552;
   1:  PR[91,3] = PR[90,3] + 58.632;
   1:L PR[91] R[100]mm/sec CNT100;
   1:  PR[91,1] = PR[90,1] + -45.662;
   1:  PR[91,2] = PR[90,2] + 20.611;
   1:  PR[91,3] = PR[90,3] + 58.647;
   1:L PR[91] R[100]mm/sec CNT100;
   1:  PR[91,1] = PR[90,1] + -46.250;
   1:  PR[91,2] = PR[90,2] + 20.657;
   1:  PR[91,3] = PR[90,3] + 58.648;
   1:L PR[91] R[100]mm/sec CNT100;
   1:  PR[91,1] = PR[90,1] + -50.365;
   1:  PR[91,2] = PR[90,2] + 21.104;
   1:  PR[91,3] = PR[90,3] + 58.650;
   1:L PR[91] R[100]mm/sec CNT100;
   1:  PR[91,1] = PR[90,1] + -52.776;
   1:  PR[91,2] = PR[90,2] + 21.328;
   1:  PR[91,3] = PR[90,3] + 58.664;
   1:L PR[91] R[100]mm/sec CNT100;
   1:  PR[91,1] = PR[90,1] + -54.749;
   1:  PR[91,2] = PR[90,2] + 21.228;
   1:  PR[91,3] = PR[90,3] + 58.672;
   1:L PR[91] R[100]mm/sec CNT100;
   1:  PR[91,1] = PR[90,1] + -59.584;
   1:  PR[91,2] = PR[90,2] + 20.927;
   1:  PR[91,3] = PR[90,3] + 58.679;
   1:L PR[91] R[100]mm/sec CNT100;
   1:  PR[91] = PR[90];
   1:  PR[91,1] = PR[90,1] + -63.300;
   1:  PR[91,2] = PR[90,2] + 20.025;
   1:  PR[91,3] = PR[90,3] + 59.995;
   1:L PR[91] R[100]mm/sec CNT100;
   1:  PR[91,1] = PR[90,1] + -64.396;
   1:  PR[91,2] = PR[90,2] + 19.758;
   1:  PR[91,3] = PR[90,3] + 58.706;
   1:L PR[91] R[100]mm/sec CNT100;
   1:  PR[91,1] = PR[90,1] + -67.203;
   1:  PR[91,2] = PR[90,2] + 18.570;
   1:  PR[91,3] = PR[90,3] + 58.710;
   1:L PR[91] R[100]mm/sec CNT100;
   1:  PR[91,1] = PR[90,1] + -69.539;
   1:  PR[91,2] = PR[90,2] + 17.553;
   1:  PR[91,3] = PR[90,3] + 58.720;
   1:L PR[91] R[100]mm/sec CNT100;
   1:  PR[91,1] = PR[90,1] + -73.874;
   1:  PR[91,2] = PR[90,2] + 14.658;
   1:  PR[91,3] = PR[90,3] + 58.729;
   1:L PR[91] R[100]mm/sec CNT100;
   1:  PR[91,1] = PR[90,1] + -76.501;
   1:  PR[91,2] = PR[90,2] + 12.037;
   1:  PR[91,3] = PR[90,3] + 58.746;
   1:L PR[91] R[100]mm/sec CNT100;
   1:  PR[91,1] = PR[90,1] + -77.202;
   1:  PR[91,2] = PR[90,2] + 11.296;
   1:  PR[91,3] = PR[90,3] + 58.759;
   1:L PR[91] R[100]mm/sec CNT100;
   1:  PR[91,1] = PR[90,1] + -79.521;
   1:  PR[91,2] = PR[90,2] + 7.522;
   1:  PR[91,3] = PR[90,3] + 58.762;
   1:L PR[91] R[100]mm/sec CNT100;
   1:  PR[91,1] = PR[90,1] + -80.934;
   1:  PR[91,2] = PR[90,2] + 3.464;
   1:  PR[91,3] = PR[90,3] + 58.777;
   1:L PR[91] R[100]mm/sec CNT100;
   1:  PR[91,1] = PR[90,1] + -81.041;
   1:  PR[91,2] = PR[90,2] + 2.531;
   1:  PR[91,3] = PR[90,3] + 58.792;
   1:L PR[91] R[100]mm/sec CNT100;
   1:  PR[91,1] = PR[90,1] + -81.224;
   1:  PR[91,2] = PR[90,2] + 1.545;
   1:  PR[91,3] = PR[90,3] + 58.795;
   1:L PR[91] R[100]mm/sec CNT100;
   1:  PR[91,1] = PR[90,1] + -81.302;
   1:  PR[91,2] = PR[90,2] + 1.004;
   1:  PR[91,3] = PR[90,3] + 58.798;
   1:L PR[91] R[100]mm/sec CNT100;
   1:  PR[91,1] = PR[90,1] + -81.500;
   1:  PR[91,2] = PR[90,2] + -0.719;
   1:  PR[91,3] = PR[90,3] + 58.800;
   1:L PR[91] R[100]mm/sec CNT100;
   1:  PR[91,1] = PR[90,1] + -81.281;
   1:  PR[91,2] = PR[90,2] + -2.474;
   1:  PR[91,3] = PR[90,3] + 58.806;
   1:L PR[91] R[100]mm/sec CNT100;
   1:  PR[91,1] = PR[90,1] + -81.026;
   1:  PR[91,2] = PR[90,2] + -3.689;
   1:  PR[91,3] = PR[90,3] + 58.812;
   1:L PR[91] R[100]mm/sec CNT100;
   1:  PR[91,1] = PR[90,1] + -80.868;
   1:  PR[91,2] = PR[90,2] + -4.986;
   1:  PR[91,3] = PR[90,3] + 58.816;
   1:L PR[91] R[100]mm/sec CNT100;
   1:  PR[91,1] = PR[90,1] + -79.888;
   1:  PR[91,2] = PR[90,2] + -7.713;
   1:  PR[91,3] = PR[90,3] + 58.820;
   1:L PR[91] R[100]mm/sec CNT100;
   1:  PR[91,1] = PR[90,1] + -79.352;
   1:  PR[91,2] = PR[90,2] + -9.133;
   1:  PR[91,3] = PR[90,3] + 58.830;
   1:L PR[91] R[100]mm/sec CNT100;
   1:  PR[91,1] = PR[90,1] + -77.963;
   1:  PR[91,2] = PR[90,2] + -11.321;
   1:  PR[91,3] = PR[90,3] + 58.835;
   1:L PR[91] R[100]mm/sec CNT100;
   1:  PR[91,1] = PR[90,1] + -76.800;
   1:  PR[91,2] = PR[90,2] + -13.052;
   1:  PR[91,3] = PR[90,3] + 58.844;
   1:L PR[91] R[100]mm/sec CNT100;
   1:  PR[91,1] = PR[90,1] + -75.336;
   1:  PR[91,2] = PR[90,2] + -14.554;
   1:  PR[91,3] = PR[90,3] + 58.851;
   1:L PR[91] R[100]mm/sec CNT100;
   1:  PR[91,1] = PR[90,1] + -73.196;
   1:  PR[91,2] = PR[90,2] + -16.594;
   1:  PR[91,3] = PR[90,3] + 58.858;
   1:L PR[91] R[100]mm/sec CNT100;
   1:  PR[91,1] = PR[90,1] + -72.088;
   1:  PR[91,2] = PR[90,2] + -17.356;
   1:  PR[91,3] = PR[90,3] + 58.868;
   1:L PR[91] R[100]mm/sec CNT100;
   1:  PR[91,1] = PR[90,1] + -68.529;
   1:  PR[91,2] = PR[90,2] + -19.573;
   1:  PR[91,3] = PR[90,3] + 58.873;
   1:L PR[91] R[100]mm/sec CNT100;
   1:  PR[91,1] = PR[90,1] + -68.295;
   1:  PR[91,2] = PR[90,2] + -19.676;
   1:  PR[91,3] = PR[90,3] + 58.887;
   1:L PR[91] R[100]mm/sec CNT100;
   1:  PR[91,1] = PR[90,1] + -66.882;
   1:  PR[91,2] = PR[90,2] + -20.213;
   1:  PR[91,3] = PR[90,3] + 58.888;
   1:L PR[91] R[100]mm/sec CNT100;
   1:  PR[91,1] = PR[90,1] + -62.978;
   1:  PR[91,2] = PR[90,2] + -21.638;
   1:  PR[91,3] = PR[90,3] + 58.893;
   1:L PR[91] R[100]mm/sec CNT100;
   1:  PR[91,1] = PR[90,1] + -60.584;
   1:  PR[91,2] = PR[90,2] + -22.094;
   1:  PR[91,3] = PR[90,3] + 58.907;
   1:L PR[91] R[100]mm/sec CNT100;
   1:  PR[91,1] = PR[90,1] + -56.792;
   1:  PR[91,2] = PR[90,2] + -22.781;
   1:  PR[91,3] = PR[90,3] + 58.915;
   1:L PR[91] R[100]mm/sec CNT100;
   1:  PR[91,1] = PR[90,1] + -51.341;
   1:  PR[91,2] = PR[90,2] + -22.894;
   1:  PR[91,3] = PR[90,3] + 58.928;
   1:L PR[91] R[100]mm/sec CNT100;
   1:  PR[91,1] = PR[90,1] + -50.303;
   1:  PR[91,2] = PR[90,2] + -22.936;
   1:  PR[91,3] = PR[90,3] + 58.946;
   1:L PR[91] R[100]mm/sec CNT100;
   1:  PR[91,1] = PR[90,1] + -49.597;
   1:  PR[91,2] = PR[90,2] + -22.905;
   1:  PR[91,3] = PR[90,3] + 58.950;
   1:L PR[91] R[100]mm/sec CNT100;
   1:  PR[91,1] = PR[90,1] + -44.748;
   1:  PR[91,2] = PR[90,2] + -22.374;
   1:  PR[91,3] = PR[90,3] + 58.952;
   1:L PR[91] R[100]mm/sec CNT100;
   1:  PR[91,1] = PR[90,1] + -39.532;
   1:  PR[91,2] = PR[90,2] + -21.374;
   1:  PR[91,3] = PR[90,3] + 58.969;
   1:L PR[91] R[100]mm/sec CNT100;
   1:  PR[91,1] = PR[90,1] + -34.393;
   1:  PR[91,2] = PR[90,2] + -19.920;
   1:  PR[91,3] = PR[90,3] + 58.986;
   1:L PR[91] R[100]mm/sec CNT100;
   1:  PR[91,1] = PR[90,1] + -29.712;
   1:  PR[91,2] = PR[90,2] + -18.229;
   1:  PR[91,3] = PR[90,3] + 59.004;
   1:L PR[91] R[100]mm/sec CNT100;
   1:  PR[91,1] = PR[90,1] + -28.170;
   1:  PR[91,2] = PR[90,2] + -17.827;
   1:  PR[91,3] = PR[90,3] + 59.021;
   1:L PR[91] R[100]mm/sec CNT100;
   1:  PR[91,1] = PR[90,1] + -26.953;
   1:  PR[91,2] = PR[90,2] + -18.630;
   1:  PR[91,3] = PR[90,3] + 59.027;
   1:L PR[91] R[100]mm/sec CNT100;
   1:  PR[91,1] = PR[90,1] + -22.517;
   1:  PR[91,2] = PR[90,2] + -21.035;
   1:  PR[91,3] = PR[90,3] + 59.032;
   1:L PR[91] R[100]mm/sec CNT100;
   1:  PR[91,1] = PR[90,1] + -22.224;
   1:  PR[91,2] = PR[90,2] + -21.161;
   1:  PR[91,3] = PR[90,3] + 59.049;
   1:L PR[91] R[100]mm/sec CNT100;
   1:  PR[91,1] = PR[90,1] + -17.803;
   1:  PR[91,2] = PR[90,2] + -22.450;
   1:  PR[91,3] = PR[90,3] + 59.050;
   1:L PR[91] R[100]mm/sec CNT100;
   1:  PR[91,1] = PR[90,1] + -16.764;
   1:  PR[91,2] = PR[90,2] + -22.727;
   1:  PR[91,3] = PR[90,3] + 59.065;
   1:L PR[91] R[100]mm/sec CNT100;
   1:  PR[91,1] = PR[90,1] + -11.099;
   1:  PR[91,2] = PR[90,2] + -23.174;
   1:  PR[91,3] = PR[90,3] + 59.069;
   1:L PR[91] R[100]mm/sec CNT100;
   1:  PR[91,1] = PR[90,1] + -8.680;
   1:  PR[91,2] = PR[90,2] + -22.870;
   1:  PR[91,3] = PR[90,3] + 59.088;
   1:L PR[91] R[100]mm/sec CNT100;
   1:  PR[91,1] = PR[90,1] + -5.504;
   1:  PR[91,2] = PR[90,2] + -22.511;
   1:  PR[91,3] = PR[90,3] + 59.096;
   1:L PR[91] R[100]mm/sec CNT100;
   1:  PR[91,1] = PR[90,1] + -0.277;
   1:  PR[91,2] = PR[90,2] + -20.808;
   1:  PR[91,3] = PR[90,3] + 59.107;
   1:L PR[91] R[100]mm/sec CNT100;
   1:  PR[91,1] = PR[90,1] + 1.131;
   1:  PR[91,2] = PR[90,2] + -19.998;
   1:  PR[91,3] = PR[90,3] + 59.125;
   1:L PR[91] R[100]mm/sec CNT100;
   1:  PR[91,1] = PR[90,1] + 5.267;
   1:  PR[91,2] = PR[90,2] + -17.868;
   1:  PR[91,3] = PR[90,3] + 59.131;
   1:L PR[91] R[100]mm/sec CNT100;
   1:  PR[91,1] = PR[90,1] + 7.580;
   1:  PR[91,2] = PR[90,2] + -19.696;
   1:  PR[91,3] = PR[90,3] + 59.147;
   1:L PR[91] R[100]mm/sec CNT100;
   1:  PR[91,1] = PR[90,1] + 9.170;
   1:  PR[91,2] = PR[90,2] + -20.679;
   1:  PR[91,3] = PR[90,3] + 59.156;
   1:L PR[91] R[100]mm/sec CNT100;
   1:  PR[91,1] = PR[90,1] + 12.463;
   1:  PR[91,2] = PR[90,2] + -22.462;
   1:  PR[91,3] = PR[90,3] + 59.163;
   1:L PR[91] R[100]mm/sec CNT100;
   1:  PR[91,1] = PR[90,1] + 14.508;
   1:  PR[91,2] = PR[90,2] + -23.102;
   1:  PR[91,3] = PR[90,3] + 59.175;
   1:L PR[91] R[100]mm/sec CNT100;
   1:  PR[91,1] = PR[90,1] + 17.807;
   1:  PR[91,2] = PR[90,2] + -24.002;
   1:  PR[91,3] = PR[90,3] + 59.183;
   1:L PR[91] R[100]mm/sec CNT100;
   1:  PR[91,1] = PR[90,1] + 20.234;
   1:  PR[91,2] = PR[90,2] + -24.135;
   1:  PR[91,3] = PR[90,3] + 59.194;
   1:L PR[91] R[100]mm/sec CNT100;
   1:  PR[91,1] = PR[90,1] + 23.391;
   1:  PR[91,2] = PR[90,2] + -24.261;
   1:  PR[91,3] = PR[90,3] + 59.202;
   1:L PR[91] R[100]mm/sec CNT100;
   1:  PR[91,1] = PR[90,1] + 26.055;
   1:  PR[91,2] = PR[90,2] + -23.742;
   1:  PR[91,3] = PR[90,3] + 59.213;
   1:L PR[91] R[100]mm/sec CNT100;
   1:  PR[91,1] = PR[90,1] + 29.010;
   1:  PR[91,2] = PR[90,2] + -23.188;
   1:  PR[91,3] = PR[90,3] + 59.222;
   1:L PR[91] R[100]mm/sec CNT100;
   1:  PR[91,1] = PR[90,1] + 29.795;
   1:  PR[91,2] = PR[90,2] + -22.934;
   1:  PR[91,3] = PR[90,3] + 59.232;
   1:L PR[91] R[100]mm/sec CNT100;
   1:  PR[91,1] = PR[90,1] + 31.201;
   1:  PR[91,2] = PR[90,2] + -22.391;
   1:  PR[91,3] = PR[90,3] + 59.235;
   1:L PR[91] R[100]mm/sec CNT100;
   1:  PR[91,1] = PR[90,1] + 32.090;
   1:  PR[91,2] = PR[90,2] + -21.977;
   1:  PR[91,3] = PR[90,3] + 59.240;
   1:L PR[91] R[100]mm/sec CNT100;
   1:  PR[91,1] = PR[90,1] + 33.063;
   1:  PR[91,2] = PR[90,2] + -22.359;
   1:  PR[91,3] = PR[90,3] + 59.243;
   1:L PR[91] R[100]mm/sec CNT100;
   1:  PR[91,1] = PR[90,1] + 34.697;
   1:  PR[91,2] = PR[90,2] + -22.864;
   1:  PR[91,3] = PR[90,3] + 59.247;
   1:L PR[91] R[100]mm/sec CNT100;
   1:  PR[91,1] = PR[90,1] + 40.455;
   1:  PR[91,2] = PR[90,2] + -24.395;
   1:  PR[91,3] = PR[90,3] + 59.253;
   1:L PR[91] R[100]mm/sec CNT100;
   1:  PR[91,1] = PR[90,1] + 44.795;
   1:  PR[91,2] = PR[90,2] + -24.961;
   1:  PR[91,3] = PR[90,3] + 59.273;
   1:L PR[91] R[100]mm/sec CNT100;
   1:  PR[91,1] = PR[90,1] + 47.535;
   1:  PR[91,2] = PR[90,2] + -25.077;
   1:  PR[91,3] = PR[90,3] + 59.287;
   1:L PR[91] R[100]mm/sec CNT100;
   1:  PR[91,1] = PR[90,1] + 49.139;
   1:  PR[91,2] = PR[90,2] + -25.169;
   1:  PR[91,3] = PR[90,3] + 59.297;
   1:L PR[91] R[100]mm/sec CNT100;
   1:  PR[91,1] = PR[90,1] + 50.670;
   1:  PR[91,2] = PR[90,2] + -25.177;
   1:  PR[91,3] = PR[90,3] + 59.302;
   1:L PR[91] R[100]mm/sec CNT100;
   1:  PR[91,1] = PR[90,1] + 54.111;
   1:  PR[91,2] = PR[90,2] + -24.975;
   1:  PR[91,3] = PR[90,3] + 59.307;
   1:L PR[91] R[100]mm/sec CNT100;
   1:  PR[91,1] = PR[90,1] + 60.632;
   1:  PR[91,2] = PR[90,2] + -23.936;
   1:  PR[91,3] = PR[90,3] + 59.319;
   1:L PR[91] R[100]mm/sec CNT100;
   1:  PR[91,1] = PR[90,1] + 64.866;
   1:  PR[91,2] = PR[90,2] + -22.446;
   1:  PR[91,3] = PR[90,3] + 59.341;
   1:L PR[91] R[100]mm/sec CNT100;
   1:  PR[91,1] = PR[90,1] + 67.173;
   1:  PR[91,2] = PR[90,2] + -21.607;
   1:  PR[91,3] = PR[90,3] + 59.356;
   1:L PR[91] R[100]mm/sec CNT100;
   1:  PR[91,1] = PR[90,1] + 69.119;
   1:  PR[91,2] = PR[90,2] + -20.476;
   1:  PR[91,3] = PR[90,3] + 59.365;
   1:L PR[91] R[100]mm/sec CNT100;
   1:  PR[91,1] = PR[90,1] + 72.652;
   1:  PR[91,2] = PR[90,2] + -18.382;
   1:  PR[91,3] = PR[90,3] + 59.372;
   1:L PR[91] R[100]mm/sec CNT100;
   1:  PR[91,1] = PR[90,1] + 75.187;
   1:  PR[91,2] = PR[90,2] + -16.098;
   1:  PR[91,3] = PR[90,3] + 59.386;
   1:L PR[91] R[100]mm/sec CNT100;
   1:  PR[91,1] = PR[90,1] + 76.734;
   1:  PR[91,2] = PR[90,2] + -14.613;
   1:  PR[91,3] = PR[90,3] + 59.397;
   1:L PR[91] R[100]mm/sec CNT100;
   1:  PR[91,1] = PR[90,1] + 76.945;
   1:  PR[91,2] = PR[90,2] + -14.322;
   1:  PR[91,3] = PR[90,3] + 59.405;
   1:L PR[91] R[100]mm/sec CNT100;
   1:  PR[91,1] = PR[90,1] + 79.574;
   1:  PR[91,2] = PR[90,2] + -10.375;
   1:  PR[91,3] = PR[90,3] + 59.406;
   1:L PR[91] R[100]mm/sec CNT100;
   1:  PR[91,1] = PR[90,1] + 80.037;
   1:  PR[91,2] = PR[90,2] + -9.230;
   1:  PR[91,3] = PR[90,3] + 59.422;
   1:L PR[91] R[100]mm/sec CNT100;
   1:  PR[91,1] = PR[90,1] + 81.364;
   1:  PR[91,2] = PR[90,2] + -5.675;
   1:  PR[91,3] = PR[90,3] + 59.426;
   1:L PR[91] R[100]mm/sec CNT100;
   1:  PR[91,1] = PR[90,1] + 81.591;
   1:  PR[91,2] = PR[90,2] + -3.957;
   1:  PR[91,3] = PR[90,3] + 59.439;
   1:L PR[91] R[100]mm/sec CNT100;
   1:  PR[91,1] = PR[90,1] + 81.945;
   1:  PR[91,2] = PR[90,2] + -2.030;
   1:  PR[91,3] = PR[90,3] + 59.445;
   1:L PR[91] R[100]mm/sec CNT100;
   1:  PR[91,1] = PR[90,1] + 82.095;
   1:  PR[91,2] = PR[90,2] + -0.804;
   1:  PR[91,3] = PR[90,3] + 59.451;
   1:L PR[91] R[100]mm/sec CNT100;
   1:  PR[91,1] = PR[90,1] + 81.751;
   1:  PR[91,2] = PR[90,2] + 0.935;
   1:  PR[91,3] = PR[90,3] + 59.455;
   1:L PR[91] R[100]mm/sec CNT100;
   1:  PR[91,1] = PR[90,1] + 81.359;
   1:  PR[91,2] = PR[90,2] + 4.234;
   1:  PR[91,3] = PR[90,3] + 59.461;
   1:L PR[91] R[100]mm/sec CNT100;
   1:  PR[91,1] = PR[90,1] + 80.030;
   1:  PR[91,2] = PR[90,2] + 7.784;
   1:  PR[91,3] = PR[90,3] + 59.473;
   1:L PR[91] R[100]mm/sec CNT100;
   1:  PR[91,1] = PR[90,1] + 79.568;
   1:  PR[91,2] = PR[90,2] + 8.927;
   1:  PR[91,3] = PR[90,3] + 59.485;
   1:L PR[91] R[100]mm/sec CNT100;
   1:  PR[91,1] = PR[90,1] + 76.927;
   1:  PR[91,2] = PR[90,2] + 12.886;
   1:  PR[91,3] = PR[90,3] + 59.489;
   1:L PR[91] R[100]mm/sec CNT100;
   1:  PR[91,1] = PR[90,1] + 76.719;
   1:  PR[91,2] = PR[90,2] + 13.172;
   1:  PR[91,3] = PR[90,3] + 59.505;
   1:L PR[91] R[100]mm/sec CNT100;
   1:  PR[91,1] = PR[90,1] + 75.188;
   1:  PR[91,2] = PR[90,2] + 14.638;
   1:  PR[91,3] = PR[90,3] + 59.507;
   1:L PR[91] R[100]mm/sec CNT100;
   1:  PR[91,1] = PR[90,1] + 72.629;
   1:  PR[91,2] = PR[90,2] + 16.940;
   1:  PR[91,3] = PR[90,3] + 59.514;
   1:L PR[91] R[100]mm/sec CNT100;
   1:  PR[91,1] = PR[90,1] + 67.154;
   1:  PR[91,2] = PR[90,2] + 20.156;
   1:  PR[91,3] = PR[90,3] + 59.525;
   1:L PR[91] R[100]mm/sec CNT100;
   1:  PR[91,1] = PR[90,1] + 64.857;
   1:  PR[91,2] = PR[90,2] + 20.987;
   1:  PR[91,3] = PR[90,3] + 59.547;
   1:L PR[91] R[100]mm/sec CNT100;
   1:  PR[91,1] = PR[90,1] + 60.651;
   1:  PR[91,2] = PR[90,2] + 22.473;
   1:  PR[91,3] = PR[90,3] + 59.555;
   1:L PR[91] R[100]mm/sec CNT100;
   1:  PR[91,1] = PR[90,1] + 54.129;
   1:  PR[91,2] = PR[90,2] + 23.516;
   1:  PR[91,3] = PR[90,3] + 59.570;
   1:L PR[91] R[100]mm/sec CNT100;
   1:  PR[91,1] = PR[90,1] + 50.683;
   1:  PR[91,2] = PR[90,2] + 23.717;
   1:  PR[91,3] = PR[90,3] + 59.592;
   1:L PR[91] R[100]mm/sec CNT100;
   1:  PR[91,1] = PR[90,1] + 49.143;
   1:  PR[91,2] = PR[90,2] + 23.711;
   1:  PR[91,3] = PR[90,3] + 59.604;
   1:L PR[91] R[100]mm/sec CNT100;
   1:  PR[91,1] = PR[90,1] + 47.536;
   1:  PR[91,2] = PR[90,2] + 23.618;
   1:  PR[91,3] = PR[90,3] + 59.609;
   1:L PR[91] R[100]mm/sec CNT100;
   1:  PR[91,1] = PR[90,1] + 44.795;
   1:  PR[91,2] = PR[90,2] + 23.502;
   1:  PR[91,3] = PR[90,3] + 59.615;
   1:L PR[91] R[100]mm/sec CNT100;
   1:  PR[91,1] = PR[90,1] + 40.455;
   1:  PR[91,2] = PR[90,2] + 22.936;
   1:  PR[91,3] = PR[90,3] + 59.624;
   1:L PR[91] R[100]mm/sec CNT100;
   1:  PR[91,1] = PR[90,1] + 34.698;
   1:  PR[91,2] = PR[90,2] + 21.405;
   1:  PR[91,3] = PR[90,3] + 59.639;
   1:L PR[91] R[100]mm/sec CNT100;
   1:  PR[91,1] = PR[90,1] + 33.063;
   1:  PR[91,2] = PR[90,2] + 20.900;
   1:  PR[91,3] = PR[90,3] + 59.659;
   1:L PR[91] R[100]mm/sec CNT100;
   1:  PR[91,1] = PR[90,1] + 32.090;
   1:  PR[91,2] = PR[90,2] + 20.518;
   1:  PR[91,3] = PR[90,3] + 59.664;
   1:L PR[91] R[100]mm/sec CNT100;
   1:  PR[91,1] = PR[90,1] + 31.201;
   1:  PR[91,2] = PR[90,2] + 20.932;
   1:  PR[91,3] = PR[90,3] + 59.668;
   1:L PR[91] R[100]mm/sec CNT100;
   1:  PR[91,1] = PR[90,1] + 29.792;
   1:  PR[91,2] = PR[90,2] + 21.476;
   1:  PR[91,3] = PR[90,3] + 59.671;
   1:L PR[91] R[100]mm/sec CNT100;
   1:  PR[91,1] = PR[90,1] + 29.101;
   1:  PR[91,2] = PR[90,2] + 21.703;
   1:  PR[91,3] = PR[90,3] + 59.676;
   1:L PR[91] R[100]mm/sec CNT100;
   1:  PR[91,1] = PR[90,1] + 26.215;
   1:  PR[91,2] = PR[90,2] + 22.276;
   1:  PR[91,3] = PR[90,3] + 59.679;
   1:L PR[91] R[100]mm/sec CNT100;
   1:  PR[91,1] = PR[90,1] + 23.400;
   1:  PR[91,2] = PR[90,2] + 22.803;
   1:  PR[91,3] = PR[90,3] + 59.689;
   1:L PR[91] R[100]mm/sec CNT100;
   1:  PR[91,1] = PR[90,1] + 20.235;
   1:  PR[91,2] = PR[90,2] + 22.676;
   1:  PR[91,3] = PR[90,3] + 59.698;
   1:L PR[91] R[100]mm/sec CNT100;
   1:  PR[91,1] = PR[90,1] + 17.809;
   1:  PR[91,2] = PR[90,2] + 22.543;
   1:  PR[91,3] = PR[90,3] + 59.709;
   1:L PR[91] R[100]mm/sec CNT100;
   1:  PR[91,1] = PR[90,1] + 14.510;
   1:  PR[91,2] = PR[90,2] + 21.644;
   1:  PR[91,3] = PR[90,3] + 59.717;
   1:L PR[91] R[100]mm/sec CNT100;
   1:  PR[91,1] = PR[90,1] + 12.466;
   1:  PR[91,2] = PR[90,2] + 21.005;
   1:  PR[91,3] = PR[90,3] + 59.729;
   1:L PR[91] R[100]mm/sec CNT100;
   1:  PR[91,1] = PR[90,1] + 9.153;
   1:  PR[91,2] = PR[90,2] + 19.209;
   1:  PR[91,3] = PR[90,3] + 59.736;
   1:L PR[91] R[100]mm/sec CNT100;
   1:  PR[91,1] = PR[90,1] + 7.592;
   1:  PR[91,2] = PR[90,2] + 18.245;
   1:  PR[91,3] = PR[90,3] + 59.749;
   1:L PR[91] R[100]mm/sec CNT100;
   1:  PR[91,1] = PR[90,1] + 5.298;
   1:  PR[91,2] = PR[90,2] + 16.350;
   1:  PR[91,3] = PR[90,3] + 59.755;
   1:L PR[91] R[100]mm/sec CNT100;
   1:  PR[91,1] = PR[90,1] + 1.074;
   1:  PR[91,2] = PR[90,2] + 18.571;
   1:  PR[91,3] = PR[90,3] + 59.765;
   1:L PR[91] R[100]mm/sec CNT100;
   1:  PR[91,1] = PR[90,1] + -0.261;
   1:  PR[91,2] = PR[90,2] + 19.342;
   1:  PR[91,3] = PR[90,3] + 59.781;
   1:L PR[91] R[100]mm/sec CNT100;
   1:  PR[91,1] = PR[90,1] + -5.494;
   1:  PR[91,2] = PR[90,2] + 21.051;
   1:  PR[91,3] = PR[90,3] + 59.786;
   1:L PR[91] R[100]mm/sec CNT100;
   1:  PR[91,1] = PR[90,1] + -7.520;
   1:  PR[91,2] = PR[90,2] + 21.304;
   1:  PR[91,3] = PR[90,3] + 59.805;
   1:L PR[91] R[100]mm/sec CNT100;
   1:  PR[91,1] = PR[90,1] + -11.064;
   1:  PR[91,2] = PR[90,2] + 21.715;
   1:  PR[91,3] = PR[90,3] + 59.811;
   1:L PR[91] R[100]mm/sec CNT100;
   1:  PR[91,1] = PR[90,1] + -16.732;
   1:  PR[91,2] = PR[90,2] + 21.274;
   1:  PR[91,3] = PR[90,3] + 59.823;
   1:L PR[91] R[100]mm/sec CNT100;
   1:  PR[91,1] = PR[90,1] + -17.777;
   1:  PR[91,2] = PR[90,2] + 20.996;
   1:  PR[91,3] = PR[90,3] + 59.843;
   1:L PR[91] R[100]mm/sec CNT100;
   1:  PR[91,1] = PR[90,1] + -22.187;
   1:  PR[91,2] = PR[90,2] + 19.717;
   1:  PR[91,3] = PR[90,3] + 59.846;
   1:L PR[91] R[100]mm/sec CNT100;
   1:  PR[91,1] = PR[90,1] + -22.490;
   1:  PR[91,2] = PR[90,2] + 19.587;
   1:  PR[91,3] = PR[90,3] + 59.862;
   1:L PR[91] R[100]mm/sec CNT100;
   1:  PR[91,1] = PR[90,1] + -26.866;
   1:  PR[91,2] = PR[90,2] + 17.226;
   1:  PR[91,3] = PR[90,3] + 59.863;
   1:L PR[91] R[100]mm/sec CNT100;
   1:  PR[91,1] = PR[90,1] + -28.299;
   1:  PR[91,2] = PR[90,2] + 16.277;
   1:  PR[91,3] = PR[90,3] + 59.880;
   1:L PR[91] R[100]mm/sec CNT100;
   1:  PR[91,1] = PR[90,1] + -29.692;
   1:  PR[91,2] = PR[90,2] + 16.842;
   1:  PR[91,3] = PR[90,3] + 59.885;
   1:L PR[91] R[100]mm/sec CNT100;
   1:  PR[91,1] = PR[90,1] + -34.610;
   1:  PR[91,2] = PR[90,2] + 18.552;
   1:  PR[91,3] = PR[90,3] + 59.890;
   1:L PR[91] R[100]mm/sec CNT100;
   1:  PR[91,1] = PR[90,1] + -37.441;
   1:  PR[91,2] = PR[90,2] + 19.193;
   1:  PR[91,3] = PR[90,3] + 59.908;
   1:L PR[91] R[100]mm/sec CNT100;
   1:  PR[91,1] = PR[90,1] + -40.190;
   1:  PR[91,2] = PR[90,2] + 20.030;
   1:  PR[91,3] = PR[90,3] + 59.918;
   1:L PR[91] R[100]mm/sec CNT100;
   1:  PR[91,1] = PR[90,1] + -42.834;
   1:  PR[91,2] = PR[90,2] + 20.640;
   1:  PR[91,3] = PR[90,3] + 59.927;
   1:L PR[91] R[100]mm/sec CNT100;
   1:  PR[91,1] = PR[90,1] + -45.093;
   1:  PR[91,2] = PR[90,2] + 20.942;
   1:  PR[91,3] = PR[90,3] + 59.937;
   1:L PR[91] R[100]mm/sec CNT100;
   1:  PR[91,1] = PR[90,1] + -47.573;
   1:  PR[91,2] = PR[90,2] + 21.136;
   1:  PR[91,3] = PR[90,3] + 59.944;
   1:L PR[91] R[100]mm/sec CNT100;
   1:  PR[91,1] = PR[90,1] + -50.038;
   1:  PR[91,2] = PR[90,2] + 21.404;
   1:  PR[91,3] = PR[90,3] + 59.953;
   1:L PR[91] R[100]mm/sec CNT100;
   1:  PR[91,1] = PR[90,1] + -51.415;
   1:  PR[91,2] = PR[90,2] + 21.532;
   1:  PR[91,3] = PR[90,3] + 59.961;
   1:L PR[91] R[100]mm/sec CNT100;
   1:  PR[91,1] = PR[90,1] + -54.434;
   1:  PR[91,2] = PR[90,2] + 21.379;
   1:  PR[91,3] = PR[90,3] + 59.966;
   1:L PR[91] R[100]mm/sec CNT100;
   1:  PR[91,1] = PR[90,1] + -58.423;
   1:  PR[91,2] = PR[90,2] + 21.128;
   1:  PR[91,3] = PR[90,3] + 59.976;
   1:L PR[91] R[100]mm/sec CNT100;
   1:  PR[91,1] = PR[90,1] + -60.071;
   1:  PR[91,2] = PR[90,2] + 20.767;
   1:  PR[91,3] = PR[90,3] + 59.989;
   1:L PR[91] R[100]mm/sec CNT100;
   1:  PR[91] = PR[90];
   1:  PR[91,1] = PR[90,1] + -63.454;
   1:  PR[91,2] = PR[90,2] + 19.936;
   1:  PR[91,3] = PR[90,3] + 61.295;
   1:L PR[91] R[100]mm/sec CNT100;
   1:  PR[91,1] = PR[90,1] + -66.951;
   1:  PR[91,2] = PR[90,2] + 18.455;
   1:  PR[91,3] = PR[90,3] + 60.001;
   1:L PR[91] R[100]mm/sec CNT100;
   1:  PR[91,1] = PR[90,1] + -68.654;
   1:  PR[91,2] = PR[90,2] + 17.714;
   1:  PR[91,3] = PR[90,3] + 60.014;
   1:L PR[91] R[100]mm/sec CNT100;
   1:  PR[91,1] = PR[90,1] + -70.562;
   1:  PR[91,2] = PR[90,2] + 16.455;
   1:  PR[91,3] = PR[90,3] + 60.020;
   1:L PR[91] R[100]mm/sec CNT100;
   1:  PR[91,1] = PR[90,1] + -73.030;
   1:  PR[91,2] = PR[90,2] + 14.797;
   1:  PR[91,3] = PR[90,3] + 60.028;
   1:L PR[91] R[100]mm/sec CNT100;
   1:  PR[91,1] = PR[90,1] + -76.495;
   1:  PR[91,2] = PR[90,2] + 11.345;
   1:  PR[91,3] = PR[90,3] + 60.038;
   1:L PR[91] R[100]mm/sec CNT100;
   1:  PR[91,1] = PR[90,1] + -78.330;
   1:  PR[91,2] = PR[90,2] + 8.532;
   1:  PR[91,3] = PR[90,3] + 60.055;
   1:L PR[91] R[100]mm/sec CNT100;
   1:  PR[91,1] = PR[90,1] + -78.923;
   1:  PR[91,2] = PR[90,2] + 7.566;
   1:  PR[91,3] = PR[90,3] + 60.066;
   1:L PR[91] R[100]mm/sec CNT100;
   1:  PR[91,1] = PR[90,1] + -80.342;
   1:  PR[91,2] = PR[90,2] + 3.486;
   1:  PR[91,3] = PR[90,3] + 60.070;
   1:L PR[91] R[100]mm/sec CNT100;
   1:  PR[91,1] = PR[90,1] + -80.380;
   1:  PR[91,2] = PR[90,2] + 3.153;
   1:  PR[91,3] = PR[90,3] + 60.085;
   1:L PR[91] R[100]mm/sec CNT100;
   1:  PR[91,1] = PR[90,1] + -80.502;
   1:  PR[91,2] = PR[90,2] + 2.433;
   1:  PR[91,3] = PR[90,3] + 60.086;
   1:L PR[91] R[100]mm/sec CNT100;
   1:  PR[91,1] = PR[90,1] + -80.864;
   1:  PR[91,2] = PR[90,2] + -0.719;
   1:  PR[91,3] = PR[90,3] + 60.088;
   1:L PR[91] R[100]mm/sec CNT100;
   1:  PR[91,1] = PR[90,1] + -80.770;
   1:  PR[91,2] = PR[90,2] + -1.472;
   1:  PR[91,3] = PR[90,3] + 60.099;
   1:L PR[91] R[100]mm/sec CNT100;
   1:  PR[91,1] = PR[90,1] + -80.414;
   1:  PR[91,2] = PR[90,2] + -3.171;
   1:  PR[91,3] = PR[90,3] + 60.102;
   1:L PR[91] R[100]mm/sec CNT100;
   1:  PR[91,1] = PR[90,1] + -80.186;
   1:  PR[91,2] = PR[90,2] + -5.042;
   1:  PR[91,3] = PR[90,3] + 60.108;
   1:L PR[91] R[100]mm/sec CNT100;
   1:  PR[91,1] = PR[90,1] + -79.381;
   1:  PR[91,2] = PR[90,2] + -7.282;
   1:  PR[91,3] = PR[90,3] + 60.114;
   1:L PR[91] R[100]mm/sec CNT100;
   1:  PR[91,1] = PR[90,1] + -78.641;
   1:  PR[91,2] = PR[90,2] + -9.241;
   1:  PR[91,3] = PR[90,3] + 60.122;
   1:L PR[91] R[100]mm/sec CNT100;
   1:  PR[91,1] = PR[90,1] + -77.535;
   1:  PR[91,2] = PR[90,2] + -10.984;
   1:  PR[91,3] = PR[90,3] + 60.129;
   1:L PR[91] R[100]mm/sec CNT100;
   1:  PR[91,1] = PR[90,1] + -76.040;
   1:  PR[91,2] = PR[90,2] + -13.208;
   1:  PR[91,3] = PR[90,3] + 60.136;
   1:L PR[91] R[100]mm/sec CNT100;
   1:  PR[91,1] = PR[90,1] + -74.964;
   1:  PR[91,2] = PR[90,2] + -14.312;
   1:  PR[91,3] = PR[90,3] + 60.145;
   1:L PR[91] R[100]mm/sec CNT100;
   1:  PR[91,1] = PR[90,1] + -72.365;
   1:  PR[91,2] = PR[90,2] + -16.790;
   1:  PR[91,3] = PR[90,3] + 60.151;
   1:L PR[91] R[100]mm/sec CNT100;
   1:  PR[91,1] = PR[90,1] + -71.751;
   1:  PR[91,2] = PR[90,2] + -17.212;
   1:  PR[91,3] = PR[90,3] + 60.163;
   1:L PR[91] R[100]mm/sec CNT100;
   1:  PR[91,1] = PR[90,1] + -68.374;
   1:  PR[91,2] = PR[90,2] + -19.315;
   1:  PR[91,3] = PR[90,3] + 60.165;
   1:L PR[91] R[100]mm/sec CNT100;
   1:  PR[91,1] = PR[90,1] + -67.674;
   1:  PR[91,2] = PR[90,2] + -19.727;
   1:  PR[91,3] = PR[90,3] + 60.179;
   1:L PR[91] R[100]mm/sec CNT100;
   1:  PR[91,1] = PR[90,1] + -67.403;
   1:  PR[91,2] = PR[90,2] + -19.828;
   1:  PR[91,3] = PR[90,3] + 60.182;
   1:L PR[91] R[100]mm/sec CNT100;
   1:  PR[91,1] = PR[90,1] + -62.006;
   1:  PR[91,2] = PR[90,2] + -21.799;
   1:  PR[91,3] = PR[90,3] + 60.183;
   1:L PR[91] R[100]mm/sec CNT100;
   1:  PR[91,1] = PR[90,1] + -57.846;
   1:  PR[91,2] = PR[90,2] + -22.590;
   1:  PR[91,3] = PR[90,3] + 60.202;
   1:L PR[91] R[100]mm/sec CNT100;
   1:  PR[91,1] = PR[90,1] + -55.779;
   1:  PR[91,2] = PR[90,2] + -22.965;
   1:  PR[91,3] = PR[90,3] + 60.217;
   1:L PR[91] R[100]mm/sec CNT100;
   1:  PR[91,1] = PR[90,1] + -52.765;
   1:  PR[91,2] = PR[90,2] + -23.027;
   1:  PR[91,3] = PR[90,3] + 60.224;
   1:L PR[91] R[100]mm/sec CNT100;
   1:  PR[91,1] = PR[90,1] + -49.526;
   1:  PR[91,2] = PR[90,2] + -23.159;
   1:  PR[91,3] = PR[90,3] + 60.234;
   1:L PR[91] R[100]mm/sec CNT100;
   1:  PR[91,1] = PR[90,1] + -47.112;
   1:  PR[91,2] = PR[90,2] + -23.052;
   1:  PR[91,3] = PR[90,3] + 60.245;
   1:L PR[91] R[100]mm/sec CNT100;
   1:  PR[91,1] = PR[90,1] + -43.996;
   1:  PR[91,2] = PR[90,2] + -22.711;
   1:  PR[91,3] = PR[90,3] + 60.253;
   1:L PR[91] R[100]mm/sec CNT100;
   1:  PR[91,1] = PR[90,1] + -40.516;
   1:  PR[91,2] = PR[90,2] + -22.044;
   1:  PR[91,3] = PR[90,3] + 60.264;
   1:L PR[91] R[100]mm/sec CNT100;
   1:  PR[91,1] = PR[90,1] + -38.576;
   1:  PR[91,2] = PR[90,2] + -21.773;
   1:  PR[91,3] = PR[90,3] + 60.276;
   1:L PR[91] R[100]mm/sec CNT100;
   1:  PR[91,1] = PR[90,1] + -36.570;
   1:  PR[91,2] = PR[90,2] + -21.377;
   1:  PR[91,3] = PR[90,3] + 60.283;
   1:L PR[91] R[100]mm/sec CNT100;
   1:  PR[91,1] = PR[90,1] + -33.458;
   1:  PR[91,2] = PR[90,2] + -20.497;
   1:  PR[91,3] = PR[90,3] + 60.290;
   1:L PR[91] R[100]mm/sec CNT100;
   1:  PR[91,1] = PR[90,1] + -30.570;
   1:  PR[91,2] = PR[90,2] + -19.454;
   1:  PR[91,3] = PR[90,3] + 60.301;
   1:L PR[91] R[100]mm/sec CNT100;
   1:  PR[91,1] = PR[90,1] + -27.006;
   1:  PR[91,2] = PR[90,2] + -18.515;
   1:  PR[91,3] = PR[90,3] + 60.311;
   1:L PR[91] R[100]mm/sec CNT100;
   1:  PR[91,1] = PR[90,1] + -22.483;
   1:  PR[91,2] = PR[90,2] + -20.979;
   1:  PR[91,3] = PR[90,3] + 60.324;
   1:L PR[91] R[100]mm/sec CNT100;
   1:  PR[91,1] = PR[90,1] + -21.542;
   1:  PR[91,2] = PR[90,2] + -21.383;
   1:  PR[91,3] = PR[90,3] + 60.341;
   1:L PR[91] R[100]mm/sec CNT100;
   1:  PR[91,1] = PR[90,1] + -17.682;
   1:  PR[91,2] = PR[90,2] + -22.508;
   1:  PR[91,3] = PR[90,3] + 60.345;
   1:L PR[91] R[100]mm/sec CNT100;
   1:  PR[91,1] = PR[90,1] + -16.101;
   1:  PR[91,2] = PR[90,2] + -22.929;
   1:  PR[91,3] = PR[90,3] + 60.358;
   1:L PR[91] R[100]mm/sec CNT100;
   1:  PR[91,1] = PR[90,1] + -10.430;
   1:  PR[91,2] = PR[90,2] + -23.375;
   1:  PR[91,3] = PR[90,3] + 60.364;
   1:L PR[91] R[100]mm/sec CNT100;
   1:  PR[91,1] = PR[90,1] + -8.625;
   1:  PR[91,2] = PR[90,2] + -23.148;
   1:  PR[91,3] = PR[90,3] + 60.383;
   1:L PR[91] R[100]mm/sec CNT100;
   1:  PR[91,1] = PR[90,1] + -4.826;
   1:  PR[91,2] = PR[90,2] + -22.718;
   1:  PR[91,3] = PR[90,3] + 60.389;
   1:L PR[91] R[100]mm/sec CNT100;
   1:  PR[91,1] = PR[90,1] + -0.866;
   1:  PR[91,2] = PR[90,2] + -21.435;
   1:  PR[91,3] = PR[90,3] + 60.402;
   1:L PR[91] R[100]mm/sec CNT100;
   1:  PR[91,1] = PR[90,1] + 0.609;
   1:  PR[91,2] = PR[90,2] + -20.996;
   1:  PR[91,3] = PR[90,3] + 60.416;
   1:L PR[91] R[100]mm/sec CNT100;
   1:  PR[91,1] = PR[90,1] + 0.827;
   1:  PR[91,2] = PR[90,2] + -20.891;
   1:  PR[91,3] = PR[90,3] + 60.422;
   1:L PR[91] R[100]mm/sec CNT100;
   1:  PR[91,1] = PR[90,1] + 5.523;
   1:  PR[91,2] = PR[90,2] + -18.457;
   1:  PR[91,3] = PR[90,3] + 60.423;
   1:L PR[91] R[100]mm/sec CNT100;
   1:  PR[91,1] = PR[90,1] + 7.438;
   1:  PR[91,2] = PR[90,2] + -19.960;
   1:  PR[91,3] = PR[90,3] + 60.441;
   1:L PR[91] R[100]mm/sec CNT100;
   1:  PR[91,1] = PR[90,1] + 8.528;
   1:  PR[91,2] = PR[90,2] + -20.634;
   1:  PR[91,3] = PR[90,3] + 60.449;
   1:L PR[91] R[100]mm/sec CNT100;
   1:  PR[91,1] = PR[90,1] + 12.341;
   1:  PR[91,2] = PR[90,2] + -22.698;
   1:  PR[91,3] = PR[90,3] + 60.453;
   1:L PR[91] R[100]mm/sec CNT100;
   1:  PR[91,1] = PR[90,1] + 13.833;
   1:  PR[91,2] = PR[90,2] + -23.165;
   1:  PR[91,3] = PR[90,3] + 60.468;
   1:L PR[91] R[100]mm/sec CNT100;
   1:  PR[91,1] = PR[90,1] + 17.687;
   1:  PR[91,2] = PR[90,2] + -24.216;
   1:  PR[91,3] = PR[90,3] + 60.473;
   1:L PR[91] R[100]mm/sec CNT100;
   1:  PR[91,1] = PR[90,1] + 19.540;
   1:  PR[91,2] = PR[90,2] + -24.318;
   1:  PR[91,3] = PR[90,3] + 60.487;
   1:L PR[91] R[100]mm/sec CNT100;
   1:  PR[91,1] = PR[90,1] + 23.268;
   1:  PR[91,2] = PR[90,2] + -24.466;
   1:  PR[91,3] = PR[90,3] + 60.493;
   1:L PR[91] R[100]mm/sec CNT100;
   1:  PR[91,1] = PR[90,1] + 25.375;
   1:  PR[91,2] = PR[90,2] + -24.056;
   1:  PR[91,3] = PR[90,3] + 60.506;
   1:L PR[91] R[100]mm/sec CNT100;
   1:  PR[91,1] = PR[90,1] + 28.883;
   1:  PR[91,2] = PR[90,2] + -23.398;
   1:  PR[91,3] = PR[90,3] + 60.513;
   1:L PR[91] R[100]mm/sec CNT100;
   1:  PR[91,1] = PR[90,1] + 29.841;
   1:  PR[91,2] = PR[90,2] + -23.088;
   1:  PR[91,3] = PR[90,3] + 60.525;
   1:L PR[91] R[100]mm/sec CNT100;
   1:  PR[91,1] = PR[90,1] + 31.454;
   1:  PR[91,2] = PR[90,2] + -22.465;
   1:  PR[91,3] = PR[90,3] + 60.529;
   1:L PR[91] R[100]mm/sec CNT100;
   1:  PR[91,1] = PR[90,1] + 33.290;
   1:  PR[91,2] = PR[90,2] + -23.031;
   1:  PR[91,3] = PR[90,3] + 60.535;
   1:L PR[91] R[100]mm/sec CNT100;
   1:  PR[91,1] = PR[90,1] + 39.169;
   1:  PR[91,2] = PR[90,2] + -24.601;
   1:  PR[91,3] = PR[90,3] + 60.541;
   1:L PR[91] R[100]mm/sec CNT100;
   1:  PR[91,1] = PR[90,1] + 44.176;
   1:  PR[91,2] = PR[90,2] + -25.252;
   1:  PR[91,3] = PR[90,3] + 60.562;
   1:L PR[91] R[100]mm/sec CNT100;
   1:  PR[91,1] = PR[90,1] + 48.562;
   1:  PR[91,2] = PR[90,2] + -25.435;
   1:  PR[91,3] = PR[90,3] + 60.579;
   1:L PR[91] R[100]mm/sec CNT100;
   1:  PR[91,1] = PR[90,1] + 53.364;
   1:  PR[91,2] = PR[90,2] + -25.153;
   1:  PR[91,3] = PR[90,3] + 60.594;
   1:L PR[91] R[100]mm/sec CNT100;
   1:  PR[91,1] = PR[90,1] + 58.718;
   1:  PR[91,2] = PR[90,2] + -24.307;
   1:  PR[91,3] = PR[90,3] + 60.610;
   1:L PR[91] R[100]mm/sec CNT100;
   1:  PR[91,1] = PR[90,1] + 59.583;
   1:  PR[91,2] = PR[90,2] + -24.147;
   1:  PR[91,3] = PR[90,3] + 60.629;
   1:L PR[91] R[100]mm/sec CNT100;
   1:  PR[91,1] = PR[90,1] + 60.843;
   1:  PR[91,2] = PR[90,2] + -23.737;
   1:  PR[91,3] = PR[90,3] + 60.632;
   1:L PR[91] R[100]mm/sec CNT100;
   1:  PR[91,1] = PR[90,1] + 64.666;
   1:  PR[91,2] = PR[90,2] + -22.392;
   1:  PR[91,3] = PR[90,3] + 60.636;
   1:L PR[91] R[100]mm/sec CNT100;
   1:  PR[91,1] = PR[90,1] + 66.211;
   1:  PR[91,2] = PR[90,2] + -21.829;
   1:  PR[91,3] = PR[90,3] + 60.650;
   1:L PR[91] R[100]mm/sec CNT100;
   1:  PR[91,1] = PR[90,1] + 68.869;
   1:  PR[91,2] = PR[90,2] + -20.284;
   1:  PR[91,3] = PR[90,3] + 60.656;
   1:L PR[91] R[100]mm/sec CNT100;
   1:  PR[91,1] = PR[90,1] + 71.760;
   1:  PR[91,2] = PR[90,2] + -18.571;
   1:  PR[91,3] = PR[90,3] + 60.666;
   1:L PR[91] R[100]mm/sec CNT100;
   1:  PR[91,1] = PR[90,1] + 76.131;
   1:  PR[91,2] = PR[90,2] + -14.636;
   1:  PR[91,3] = PR[90,3] + 60.677;
   1:L PR[91] R[100]mm/sec CNT100;
   1:  PR[91,1] = PR[90,1] + 76.822;
   1:  PR[91,2] = PR[90,2] + -13.666;
   1:  PR[91,3] = PR[90,3] + 60.697;
   1:L PR[91] R[100]mm/sec CNT100;
   1:  PR[91,1] = PR[90,1] + 79.020;
   1:  PR[91,2] = PR[90,2] + -10.365;
   1:  PR[91,3] = PR[90,3] + 60.701;
   1:L PR[91] R[100]mm/sec CNT100;
   1:  PR[91,1] = PR[90,1] + 79.200;
   1:  PR[91,2] = PR[90,2] + -9.920;
   1:  PR[91,3] = PR[90,3] + 60.715;
   1:L PR[91] R[100]mm/sec CNT100;
   1:  PR[91,1] = PR[90,1] + 80.788;
   1:  PR[91,2] = PR[90,2] + -5.668;
   1:  PR[91,3] = PR[90,3] + 60.717;
   1:L PR[91] R[100]mm/sec CNT100;
   1:  PR[91,1] = PR[90,1] + 80.923;
   1:  PR[91,2] = PR[90,2] + -4.648;
   1:  PR[91,3] = PR[90,3] + 60.732;
   1:L PR[91] R[100]mm/sec CNT100;
   1:  PR[91,1] = PR[90,1] + 81.145;
   1:  PR[91,2] = PR[90,2] + -3.435;
   1:  PR[91,3] = PR[90,3] + 60.736;
   1:L PR[91] R[100]mm/sec CNT100;
   1:  PR[91,1] = PR[90,1] + 81.467;
   1:  PR[91,2] = PR[90,2] + -0.804;
   1:  PR[91,3] = PR[90,3] + 60.740;
   1:L PR[91] R[100]mm/sec CNT100;
   1:  PR[91,1] = PR[90,1] + 81.250;
   1:  PR[91,2] = PR[90,2] + 0.292;
   1:  PR[91,3] = PR[90,3] + 60.749;
   1:L PR[91] R[100]mm/sec CNT100;
   1:  PR[91,1] = PR[90,1] + 80.782;
   1:  PR[91,2] = PR[90,2] + 4.227;
   1:  PR[91,3] = PR[90,3] + 60.753;
   1:L PR[91] R[100]mm/sec CNT100;
   1:  PR[91,1] = PR[90,1] + 79.192;
   1:  PR[91,2] = PR[90,2] + 8.477;
   1:  PR[91,3] = PR[90,3] + 60.766;
   1:L PR[91] R[100]mm/sec CNT100;
   1:  PR[91,1] = PR[90,1] + 79.013;
   1:  PR[91,2] = PR[90,2] + 8.919;
   1:  PR[91,3] = PR[90,3] + 60.781;
   1:L PR[91] R[100]mm/sec CNT100;
   1:  PR[91,1] = PR[90,1] + 76.823;
   1:  PR[91,2] = PR[90,2] + 12.203;
   1:  PR[91,3] = PR[90,3] + 60.783;
   1:L PR[91] R[100]mm/sec CNT100;
   1:  PR[91,1] = PR[90,1] + 76.114;
   1:  PR[91,2] = PR[90,2] + 13.196;
   1:  PR[91,3] = PR[90,3] + 60.797;
   1:L PR[91] R[100]mm/sec CNT100;
   1:  PR[91,1] = PR[90,1] + 71.745;
   1:  PR[91,2] = PR[90,2] + 17.123;
   1:  PR[91,3] = PR[90,3] + 60.801;
   1:L PR[91] R[100]mm/sec CNT100;
   1:  PR[91,1] = PR[90,1] + 66.209;
   1:  PR[91,2] = PR[90,2] + 20.371;
   1:  PR[91,3] = PR[90,3] + 60.821;
   1:L PR[91] R[100]mm/sec CNT100;
   1:  PR[91,1] = PR[90,1] + 60.840;
   1:  PR[91,2] = PR[90,2] + 22.281;
   1:  PR[91,3] = PR[90,3] + 60.842;
   1:L PR[91] R[100]mm/sec CNT100;
   1:  PR[91,1] = PR[90,1] + 59.608;
   1:  PR[91,2] = PR[90,2] + 22.683;
   1:  PR[91,3] = PR[90,3] + 60.862;
   1:L PR[91] R[100]mm/sec CNT100;
   1:  PR[91,1] = PR[90,1] + 58.758;
   1:  PR[91,2] = PR[90,2] + 22.840;
   1:  PR[91,3] = PR[90,3] + 60.866;
   1:L PR[91] R[100]mm/sec CNT100;
   1:  PR[91,1] = PR[90,1] + 53.376;
   1:  PR[91,2] = PR[90,2] + 23.694;
   1:  PR[91,3] = PR[90,3] + 60.869;
   1:L PR[91] R[100]mm/sec CNT100;
   1:  PR[91,1] = PR[90,1] + 48.562;
   1:  PR[91,2] = PR[90,2] + 23.976;
   1:  PR[91,3] = PR[90,3] + 60.888;
   1:L PR[91] R[100]mm/sec CNT100;
   1:  PR[91,1] = PR[90,1] + 44.176;
   1:  PR[91,2] = PR[90,2] + 23.793;
   1:  PR[91,3] = PR[90,3] + 60.904;
   1:L PR[91] R[100]mm/sec CNT100;
   1:  PR[91,1] = PR[90,1] + 39.165;
   1:  PR[91,2] = PR[90,2] + 23.142;
   1:  PR[91,3] = PR[90,3] + 60.919;
   1:L PR[91] R[100]mm/sec CNT100;
   1:  PR[91,1] = PR[90,1] + 36.437;
   1:  PR[91,2] = PR[90,2] + 22.424;
   1:  PR[91,3] = PR[90,3] + 60.936;
   1:L PR[91] R[100]mm/sec CNT100;
   1:  PR[91,1] = PR[90,1] + 33.293;
   1:  PR[91,2] = PR[90,2] + 21.573;
   1:  PR[91,3] = PR[90,3] + 60.946;
   1:L PR[91] R[100]mm/sec CNT100;
   1:  PR[91,1] = PR[90,1] + 31.454;
   1:  PR[91,2] = PR[90,2] + 21.006;
   1:  PR[91,3] = PR[90,3] + 60.957;
   1:L PR[91] R[100]mm/sec CNT100;
   1:  PR[91,1] = PR[90,1] + 29.838;
   1:  PR[91,2] = PR[90,2] + 21.631;
   1:  PR[91,3] = PR[90,3] + 60.963;
   1:L PR[91] R[100]mm/sec CNT100;
   1:  PR[91,1] = PR[90,1] + 28.991;
   1:  PR[91,2] = PR[90,2] + 21.908;
   1:  PR[91,3] = PR[90,3] + 60.969;
   1:L PR[91] R[100]mm/sec CNT100;
   1:  PR[91,1] = PR[90,1] + 26.603;
   1:  PR[91,2] = PR[90,2] + 22.385;
   1:  PR[91,3] = PR[90,3] + 60.972;
   1:L PR[91] R[100]mm/sec CNT100;
   1:  PR[91,1] = PR[90,1] + 23.278;
   1:  PR[91,2] = PR[90,2] + 23.008;
   1:  PR[91,3] = PR[90,3] + 60.981;
   1:L PR[91] R[100]mm/sec CNT100;
   1:  PR[91,1] = PR[90,1] + 19.541;
   1:  PR[91,2] = PR[90,2] + 22.859;
   1:  PR[91,3] = PR[90,3] + 60.992;
   1:L PR[91] R[100]mm/sec CNT100;
   1:  PR[91,1] = PR[90,1] + 17.689;
   1:  PR[91,2] = PR[90,2] + 22.757;
   1:  PR[91,3] = PR[90,3] + 61.005;
   1:L PR[91] R[100]mm/sec CNT100;
   1:  PR[91,1] = PR[90,1] + 13.834;
   1:  PR[91,2] = PR[90,2] + 21.706;
   1:  PR[91,3] = PR[90,3] + 61.011;
   1:L PR[91] R[100]mm/sec CNT100;
   1:  PR[91,1] = PR[90,1] + 12.342;
   1:  PR[91,2] = PR[90,2] + 21.240;
   1:  PR[91,3] = PR[90,3] + 61.025;
   1:L PR[91] R[100]mm/sec CNT100;
   1:  PR[91,1] = PR[90,1] + 8.507;
   1:  PR[91,2] = PR[90,2] + 19.161;
   1:  PR[91,3] = PR[90,3] + 61.030;
   1:L PR[91] R[100]mm/sec CNT100;
   1:  PR[91,1] = PR[90,1] + 7.451;
   1:  PR[91,2] = PR[90,2] + 18.509;
   1:  PR[91,3] = PR[90,3] + 61.045;
   1:L PR[91] R[100]mm/sec CNT100;
   1:  PR[91,1] = PR[90,1] + 5.559;
   1:  PR[91,2] = PR[90,2] + 16.946;
   1:  PR[91,3] = PR[90,3] + 61.049;
   1:L PR[91] R[100]mm/sec CNT100;
   1:  PR[91,1] = PR[90,1] + 0.849;
   1:  PR[91,2] = PR[90,2] + 19.422;
   1:  PR[91,3] = PR[90,3] + 61.057;
   1:L PR[91] R[100]mm/sec CNT100;
   1:  PR[91,1] = PR[90,1] + 0.622;
   1:  PR[91,2] = PR[90,2] + 19.532;
   1:  PR[91,3] = PR[90,3] + 61.076;
   1:L PR[91] R[100]mm/sec CNT100;
   1:  PR[91,1] = PR[90,1] + -0.867;
   1:  PR[91,2] = PR[90,2] + 19.976;
   1:L PR[91] R[100]mm/sec CNT100;
   1:  PR[91,1] = PR[90,1] + -4.812;
   1:  PR[91,2] = PR[90,2] + 21.257;
   1:  PR[91,3] = PR[90,3] + 61.082;
   1:L PR[91] R[100]mm/sec CNT100;
   1:  PR[91,1] = PR[90,1] + -10.400;
   1:  PR[91,2] = PR[90,2] + 21.916;
   1:  PR[91,3] = PR[90,3] + 61.096;
   1:L PR[91] R[100]mm/sec CNT100;
   1:  PR[91,1] = PR[90,1] + -16.073;
   1:  PR[91,2] = PR[90,2] + 21.475;
   1:  PR[91,3] = PR[90,3] + 61.115;
   1:L PR[91] R[100]mm/sec CNT100;
   1:  PR[91,1] = PR[90,1] + -17.660;
   1:  PR[91,2] = PR[90,2] + 21.053;
   1:  PR[91,3] = PR[90,3] + 61.134;
   1:L PR[91] R[100]mm/sec CNT100;
   1:  PR[91,1] = PR[90,1] + -21.511;
   1:  PR[91,2] = PR[90,2] + 19.937;
   1:  PR[91,3] = PR[90,3] + 61.140;
   1:L PR[91] R[100]mm/sec CNT100;
   1:  PR[91,1] = PR[90,1] + -22.464;
   1:  PR[91,2] = PR[90,2] + 19.528;
   1:  PR[91,3] = PR[90,3] + 61.154;
   1:L PR[91] R[100]mm/sec CNT100;
   1:  PR[91,1] = PR[90,1] + -27.004;
   1:  PR[91,2] = PR[90,2] + 17.068;
   1:  PR[91,3] = PR[90,3] + 61.157;
   1:L PR[91] R[100]mm/sec CNT100;
   1:  PR[91,1] = PR[90,1] + -29.660;
   1:  PR[91,2] = PR[90,2] + 17.729;
   1:  PR[91,3] = PR[90,3] + 61.175;
   1:L PR[91] R[100]mm/sec CNT100;
   1:  PR[91,1] = PR[90,1] + -33.547;
   1:  PR[91,2] = PR[90,2] + 19.080;
   1:  PR[91,3] = PR[90,3] + 61.184;
   1:L PR[91] R[100]mm/sec CNT100;
   1:  PR[91,1] = PR[90,1] + -38.500;
   1:  PR[91,2] = PR[90,2] + 20.202;
   1:  PR[91,3] = PR[90,3] + 61.198;
   1:L PR[91] R[100]mm/sec CNT100;
   1:  PR[91,1] = PR[90,1] + -39.544;
   1:  PR[91,2] = PR[90,2] + 20.520;
   1:  PR[91,3] = PR[90,3] + 61.215;
   1:L PR[91] R[100]mm/sec CNT100;
   1:  PR[91,1] = PR[90,1] + -40.448;
   1:  PR[91,2] = PR[90,2] + 20.729;
   1:  PR[91,3] = PR[90,3] + 61.219;
   1:L PR[91] R[100]mm/sec CNT100;
   1:  PR[91,1] = PR[90,1] + -44.524;
   1:  PR[91,2] = PR[90,2] + 21.274;
   1:  PR[91,3] = PR[90,3] + 61.222;
   1:L PR[91] R[100]mm/sec CNT100;
   1:  PR[91,1] = PR[90,1] + -48.890;
   1:  PR[91,2] = PR[90,2] + 21.614;
   1:  PR[91,3] = PR[90,3] + 61.236;
   1:L PR[91] R[100]mm/sec CNT100;
   1:  PR[91,1] = PR[90,1] + -50.063;
   1:  PR[91,2] = PR[90,2] + 21.735;
   1:  PR[91,3] = PR[90,3] + 61.251;
   1:L PR[91] R[100]mm/sec CNT100;
   1:  PR[91,1] = PR[90,1] + -54.120;
   1:  PR[91,2] = PR[90,2] + 21.529;
   1:  PR[91,3] = PR[90,3] + 61.255;
   1:L PR[91] R[100]mm/sec CNT100;
   1:  PR[91,1] = PR[90,1] + -57.159;
   1:  PR[91,2] = PR[90,2] + 21.338;
   1:  PR[91,3] = PR[90,3] + 61.269;
   1:L PR[91] R[100]mm/sec CNT100;
   1:  PR[91,1] = PR[90,1] + -61.720;
   1:  PR[91,2] = PR[90,2] + 20.341;
   1:  PR[91,3] = PR[90,3] + 61.279;
   1:L PR[91] R[100]mm/sec CNT100;
   1:  PR[91] = PR[90];
   1:  PR[91,1] = PR[90,1] + -63.055;
   1:  PR[91,2] = PR[90,2] + 19.883;
   1:  PR[91,3] = PR[90,3] + 62.595;
   1:L PR[91] R[100]mm/sec CNT100;
   1:  PR[91,1] = PR[90,1] + -66.700;
   1:  PR[91,2] = PR[90,2] + 18.341;
   1:  PR[91,3] = PR[90,3] + 61.297;
   1:L PR[91] R[100]mm/sec CNT100;
   1:  PR[91,1] = PR[90,1] + -67.764;
   1:  PR[91,2] = PR[90,2] + 17.877;
   1:  PR[91,3] = PR[90,3] + 61.311;
   1:L PR[91] R[100]mm/sec CNT100;
   1:  PR[91,1] = PR[90,1] + -70.261;
   1:  PR[91,2] = PR[90,2] + 16.230;
   1:  PR[91,3] = PR[90,3] + 61.315;
   1:L PR[91] R[100]mm/sec CNT100;
   1:  PR[91,1] = PR[90,1] + -72.189;
   1:  PR[91,2] = PR[90,2] + 14.935;
   1:  PR[91,3] = PR[90,3] + 61.325;
   1:L PR[91] R[100]mm/sec CNT100;
   1:  PR[91,1] = PR[90,1] + -75.691;
   1:  PR[91,2] = PR[90,2] + 11.451;
   1:  PR[91,3] = PR[90,3] + 61.333;
   1:L PR[91] R[100]mm/sec CNT100;
   1:  PR[91,1] = PR[90,1] + -78.212;
   1:  PR[91,2] = PR[90,2] + 7.588;
   1:  PR[91,3] = PR[90,3] + 61.350;
   1:L PR[91] R[100]mm/sec CNT100;
   1:  PR[91,1] = PR[90,1] + -79.727;
   1:  PR[91,2] = PR[90,2] + 3.487;
   1:  PR[91,3] = PR[90,3] + 61.366;
   1:L PR[91] R[100]mm/sec CNT100;
   1:  PR[91,1] = PR[90,1] + -80.218;
   1:  PR[91,2] = PR[90,2] + -0.643;
   1:  PR[91,3] = PR[90,3] + 61.381;
   1:L PR[91] R[100]mm/sec CNT100;
   1:  PR[91,1] = PR[90,1] + -79.802;
   1:  PR[91,2] = PR[90,2] + -2.655;
   1:  PR[91,3] = PR[90,3] + 61.395;
   1:L PR[91] R[100]mm/sec CNT100;
   1:  PR[91,1] = PR[90,1] + -79.504;
   1:  PR[91,2] = PR[90,2] + -5.097;
   1:  PR[91,3] = PR[90,3] + 61.402;
   1:L PR[91] R[100]mm/sec CNT100;
   1:  PR[91,1] = PR[90,1] + -78.873;
   1:  PR[91,2] = PR[90,2] + -6.852;
   1:  PR[91,3] = PR[90,3] + 61.410;
   1:L PR[91] R[100]mm/sec CNT100;
   1:  PR[91,1] = PR[90,1] + -77.930;
   1:  PR[91,2] = PR[90,2] + -9.349;
   1:  PR[91,3] = PR[90,3] + 61.417;
   1:L PR[91] R[100]mm/sec CNT100;
   1:  PR[91,1] = PR[90,1] + -77.107;
   1:  PR[91,2] = PR[90,2] + -10.646;
   1:  PR[91,3] = PR[90,3] + 61.426;
   1:L PR[91] R[100]mm/sec CNT100;
   1:  PR[91,1] = PR[90,1] + -75.280;
   1:  PR[91,2] = PR[90,2] + -13.365;
   1:  PR[91,3] = PR[90,3] + 61.431;
   1:L PR[91] R[100]mm/sec CNT100;
   1:  PR[91,1] = PR[90,1] + -74.592;
   1:  PR[91,2] = PR[90,2] + -14.070;
   1:  PR[91,3] = PR[90,3] + 61.443;
   1:L PR[91] R[100]mm/sec CNT100;
   1:  PR[91,1] = PR[90,1] + -71.535;
   1:  PR[91,2] = PR[90,2] + -16.985;
   1:  PR[91,3] = PR[90,3] + 61.446;
   1:L PR[91] R[100]mm/sec CNT100;
   1:  PR[91,1] = PR[90,1] + -71.414;
   1:  PR[91,2] = PR[90,2] + -17.068;
   1:  PR[91,3] = PR[90,3] + 61.460;
   1:L PR[91] R[100]mm/sec CNT100;
   1:  PR[91,1] = PR[90,1] + -70.202;
   1:  PR[91,2] = PR[90,2] + -17.823;
   1:  PR[91,3] = PR[90,3] + 61.461;
   1:L PR[91] R[100]mm/sec CNT100;
   1:  PR[91,1] = PR[90,1] + -66.734;
   1:  PR[91,2] = PR[90,2] + -19.862;
   1:  PR[91,3] = PR[90,3] + 61.466;
   1:L PR[91] R[100]mm/sec CNT100;
   1:  PR[91,1] = PR[90,1] + -65.059;
   1:  PR[91,2] = PR[90,2] + -20.490;
   1:  PR[91,3] = PR[90,3] + 61.480;
   1:L PR[91] R[100]mm/sec CNT100;
   1:  PR[91,1] = PR[90,1] + -61.034;
   1:  PR[91,2] = PR[90,2] + -21.959;
   1:  PR[91,3] = PR[90,3] + 61.486;
   1:L PR[91] R[100]mm/sec CNT100;
   1:  PR[91,1] = PR[90,1] + -54.758;
   1:  PR[91,2] = PR[90,2] + -23.149;
   1:  PR[91,3] = PR[90,3] + 61.500;
   1:L PR[91] R[100]mm/sec CNT100;
   1:  PR[91,1] = PR[90,1] + -54.189;
   1:  PR[91,2] = PR[90,2] + -23.161;
   1:  PR[91,3] = PR[90,3] + 61.522;
   1:L PR[91] R[100]mm/sec CNT100;
   1:  PR[91,1] = PR[90,1] + -48.748;
   1:  PR[91,2] = PR[90,2] + -23.382;
   1:  PR[91,3] = PR[90,3] + 61.524;
   1:L PR[91] R[100]mm/sec CNT100;
   1:  PR[91,1] = PR[90,1] + -44.626;
   1:  PR[91,2] = PR[90,2] + -23.200;
   1:  PR[91,3] = PR[90,3] + 61.543;
   1:L PR[91] R[100]mm/sec CNT100;
   1:  PR[91,1] = PR[90,1] + -43.244;
   1:  PR[91,2] = PR[90,2] + -23.048;
   1:  PR[91,3] = PR[90,3] + 61.557;
   1:L PR[91] R[100]mm/sec CNT100;
   1:  PR[91,1] = PR[90,1] + -41.630;
   1:  PR[91,2] = PR[90,2] + -22.739;
   1:  PR[91,3] = PR[90,3] + 61.562;
   1:L PR[91] R[100]mm/sec CNT100;
   1:  PR[91,1] = PR[90,1] + -37.746;
   1:  PR[91,2] = PR[90,2] + -22.196;
   1:  PR[91,3] = PR[90,3] + 61.568;
   1:L PR[91] R[100]mm/sec CNT100;
   1:  PR[91,1] = PR[90,1] + -33.602;
   1:  PR[91,2] = PR[90,2] + -21.379;
   1:  PR[91,3] = PR[90,3] + 61.581;
   1:L PR[91] R[100]mm/sec CNT100;
   1:  PR[91,1] = PR[90,1] + -32.523;
   1:  PR[91,2] = PR[90,2] + -21.074;
   1:  PR[91,3] = PR[90,3] + 61.596;
   1:L PR[91] R[100]mm/sec CNT100;
   1:  PR[91,1] = PR[90,1] + -31.427;
   1:  PR[91,2] = PR[90,2] + -20.678;
   1:  PR[91,3] = PR[90,3] + 61.599;
   1:L PR[91] R[100]mm/sec CNT100;
   1:  PR[91,1] = PR[90,1] + -25.692;
   1:  PR[91,2] = PR[90,2] + -19.156;
   1:  PR[91,3] = PR[90,3] + 61.603;
   1:L PR[91] R[100]mm/sec CNT100;
   1:  PR[91,1] = PR[90,1] + -22.451;
   1:  PR[91,2] = PR[90,2] + -20.922;
   1:  PR[91,3] = PR[90,3] + 61.624;
   1:L PR[91] R[100]mm/sec CNT100;
   1:  PR[91,1] = PR[90,1] + -20.861;
   1:  PR[91,2] = PR[90,2] + -21.604;
   1:  PR[91,3] = PR[90,3] + 61.636;
   1:L PR[91] R[100]mm/sec CNT100;
   1:  PR[91,1] = PR[90,1] + -17.562;
   1:  PR[91,2] = PR[90,2] + -22.566;
   1:  PR[91,3] = PR[90,3] + 61.642;
   1:L PR[91] R[100]mm/sec CNT100;
   1:  PR[91,1] = PR[90,1] + -15.438;
   1:  PR[91,2] = PR[90,2] + -23.132;
   1:  PR[91,3] = PR[90,3] + 61.654;
   1:L PR[91] R[100]mm/sec CNT100;
   1:  PR[91,1] = PR[90,1] + -9.760;
   1:  PR[91,2] = PR[90,2] + -23.576;
   1:  PR[91,3] = PR[90,3] + 61.662;
   1:L PR[91] R[100]mm/sec CNT100;
   1:  PR[91,1] = PR[90,1] + -8.571;
   1:  PR[91,2] = PR[90,2] + -23.426;
   1:  PR[91,3] = PR[90,3] + 61.681;
   1:L PR[91] R[100]mm/sec CNT100;
   1:  PR[91,1] = PR[90,1] + -4.149;
   1:  PR[91,2] = PR[90,2] + -22.926;
   1:  PR[91,3] = PR[90,3] + 61.685;
   1:L PR[91] R[100]mm/sec CNT100;
   1:  PR[91,1] = PR[90,1] + -3.315;
   1:  PR[91,2] = PR[90,2] + -22.656;
   1:  PR[91,3] = PR[90,3] + 61.701;
   1:L PR[91] R[100]mm/sec CNT100;
   1:  PR[91,1] = PR[90,1] + 1.514;
   1:  PR[91,2] = PR[90,2] + -21.221;
   1:  PR[91,3] = PR[90,3] + 61.704;
   1:L PR[91] R[100]mm/sec CNT100;
   1:  PR[91,1] = PR[90,1] + 2.553;
   1:  PR[91,2] = PR[90,2] + -20.717;
   1:  PR[91,3] = PR[90,3] + 61.721;
   1:L PR[91] R[100]mm/sec CNT100;
   1:  PR[91,1] = PR[90,1] + 5.789;
   1:  PR[91,2] = PR[90,2] + -19.040;
   1:  PR[91,3] = PR[90,3] + 61.725;
   1:L PR[91] R[100]mm/sec CNT100;
   1:  PR[91,1] = PR[90,1] + 7.299;
   1:  PR[91,2] = PR[90,2] + -20.225;
   1:  PR[91,3] = PR[90,3] + 61.737;
   1:L PR[91] R[100]mm/sec CNT100;
   1:  PR[91,1] = PR[90,1] + 7.885;
   1:  PR[91,2] = PR[90,2] + -20.588;
   1:  PR[91,3] = PR[90,3] + 61.744;
   1:L PR[91] R[100]mm/sec CNT100;
   1:  PR[91,1] = PR[90,1] + 12.218;
   1:  PR[91,2] = PR[90,2] + -22.933;
   1:  PR[91,3] = PR[90,3] + 61.746;
   1:L PR[91] R[100]mm/sec CNT100;
   1:  PR[91,1] = PR[90,1] + 13.157;
   1:  PR[91,2] = PR[90,2] + -23.227;
   1:  PR[91,3] = PR[90,3] + 61.763;
   1:L PR[91] R[100]mm/sec CNT100;
   1:  PR[91,1] = PR[90,1] + 17.567;
   1:  PR[91,2] = PR[90,2] + -24.429;
   1:  PR[91,3] = PR[90,3] + 61.767;
   1:L PR[91] R[100]mm/sec CNT100;
   1:  PR[91,1] = PR[90,1] + 18.846;
   1:  PR[91,2] = PR[90,2] + -24.500;
   1:  PR[91,3] = PR[90,3] + 61.782;
   1:L PR[91] R[100]mm/sec CNT100;
   1:  PR[91,1] = PR[90,1] + 23.151;
   1:  PR[91,2] = PR[90,2] + -24.672;
   1:  PR[91,3] = PR[90,3] + 61.787;
   1:L PR[91] R[100]mm/sec CNT100;
   1:  PR[91,1] = PR[90,1] + 28.753;
   1:  PR[91,2] = PR[90,2] + -23.609;
   1:  PR[91,3] = PR[90,3] + 61.802;
   1:L PR[91] R[100]mm/sec CNT100;
   1:  PR[91,1] = PR[90,1] + 29.887;
   1:  PR[91,2] = PR[90,2] + -23.242;
   1:  PR[91,3] = PR[90,3] + 61.821;
   1:L PR[91] R[100]mm/sec CNT100;
   1:  PR[91,1] = PR[90,1] + 30.835;
   1:  PR[91,2] = PR[90,2] + -22.876;
   1:  PR[91,3] = PR[90,3] + 61.825;
   1:L PR[91] R[100]mm/sec CNT100;
   1:  PR[91,1] = PR[90,1] + 31.882;
   1:  PR[91,2] = PR[90,2] + -23.199;
   1:  PR[91,3] = PR[90,3] + 61.829;
   1:L PR[91] R[100]mm/sec CNT100;
   1:  PR[91,1] = PR[90,1] + 37.882;
   1:  PR[91,2] = PR[90,2] + -24.807;
   1:  PR[91,3] = PR[90,3] + 61.832;
   1:L PR[91] R[100]mm/sec CNT100;
   1:  PR[91,1] = PR[90,1] + 43.559;
   1:  PR[91,2] = PR[90,2] + -25.543;
   1:  PR[91,3] = PR[90,3] + 61.854;
   1:L PR[91] R[100]mm/sec CNT100;
   1:  PR[91,1] = PR[90,1] + 43.942;
   1:  PR[91,2] = PR[90,2] + -25.559;
   1:  PR[91,3] = PR[90,3] + 61.873;
   1:L PR[91] R[100]mm/sec CNT100;
   1:  PR[91,1] = PR[90,1] + 47.890;
   1:  PR[91,2] = PR[90,2] + -25.632;
   1:  PR[91,3] = PR[90,3] + 61.875;
   1:L PR[91] R[100]mm/sec CNT100;
   1:  PR[91,1] = PR[90,1] + 49.696;
   1:  PR[91,2] = PR[90,2] + -25.502;
   1:  PR[91,3] = PR[90,3] + 61.888;
   1:L PR[91] R[100]mm/sec CNT100;
   1:  PR[91,1] = PR[90,1] + 52.615;
   1:  PR[91,2] = PR[90,2] + -25.331;
   1:  PR[91,3] = PR[90,3] + 61.894;
   1:L PR[91] R[100]mm/sec CNT100;
   1:  PR[91,1] = PR[90,1] + 55.818;
   1:  PR[91,2] = PR[90,2] + -24.825;
   1:  PR[91,3] = PR[90,3] + 61.904;
   1:L PR[91] R[100]mm/sec CNT100;
   1:  PR[91,1] = PR[90,1] + 58.533;
   1:  PR[91,2] = PR[90,2] + -24.324;
   1:  PR[91,3] = PR[90,3] + 61.916;
   1:L PR[91] R[100]mm/sec CNT100;
   1:  PR[91,1] = PR[90,1] + 62.349;
   1:  PR[91,2] = PR[90,2] + -23.082;
   1:  PR[91,3] = PR[90,3] + 61.925;
   1:L PR[91] R[100]mm/sec CNT100;
   1:  PR[91,1] = PR[90,1] + 65.255;
   1:  PR[91,2] = PR[90,2] + -22.048;
   1:  PR[91,3] = PR[90,3] + 61.939;
   1:L PR[91] R[100]mm/sec CNT100;
   1:  PR[91,1] = PR[90,1] + 68.620;
   1:  PR[91,2] = PR[90,2] + -20.093;
   1:  PR[91,3] = PR[90,3] + 61.949;
   1:L PR[91] R[100]mm/sec CNT100;
   1:  PR[91,1] = PR[90,1] + 70.870;
   1:  PR[91,2] = PR[90,2] + -18.760;
   1:  PR[91,3] = PR[90,3] + 61.963;
   1:L PR[91] R[100]mm/sec CNT100;
   1:  PR[91,1] = PR[90,1] + 75.294;
   1:  PR[91,2] = PR[90,2] + -14.783;
   1:  PR[91,3] = PR[90,3] + 61.972;
   1:L PR[91] R[100]mm/sec CNT100;
   1:  PR[91,1] = PR[90,1] + 78.449;
   1:  PR[91,2] = PR[90,2] + -10.353;
   1:  PR[91,3] = PR[90,3] + 61.992;
   1:L PR[91] R[100]mm/sec CNT100;
   1:  PR[91,1] = PR[90,1] + 80.212;
   1:  PR[91,2] = PR[90,2] + -5.659;
   1:  PR[91,3] = PR[90,3] + 62.011;
   1:L PR[91] R[100]mm/sec CNT100;
   1:  PR[91,1] = PR[90,1] + 80.254;
   1:  PR[91,2] = PR[90,2] + -5.339;
   1:  PR[91,3] = PR[90,3] + 62.028;
   1:L PR[91] R[100]mm/sec CNT100;
   1:  PR[91,1] = PR[90,1] + 80.346;
   1:  PR[91,2] = PR[90,2] + -4.839;
   1:  PR[91,3] = PR[90,3] + 62.029;
   1:L PR[91] R[100]mm/sec CNT100;
   1:  PR[91,1] = PR[90,1] + 80.839;
   1:  PR[91,2] = PR[90,2] + -0.804;
   1:  PR[91,3] = PR[90,3] + 62.031;
   1:L PR[91] R[100]mm/sec CNT100;
   1:  PR[91,1] = PR[90,1] + 80.749;
   1:  PR[91,2] = PR[90,2] + -0.351;
   1:  PR[91,3] = PR[90,3] + 62.045;
   1:L PR[91] R[100]mm/sec CNT100;
   1:  PR[91,1] = PR[90,1] + 80.205;
   1:  PR[91,2] = PR[90,2] + 4.219;
   1:  PR[91,3] = PR[90,3] + 62.046;
   1:L PR[91] R[100]mm/sec CNT100;
   1:  PR[91,1] = PR[90,1] + 78.440;
   1:  PR[91,2] = PR[90,2] + 8.909;
   1:  PR[91,3] = PR[90,3] + 62.062;
   1:L PR[91] R[100]mm/sec CNT100;
   1:  PR[91,1] = PR[90,1] + 75.280;
   1:  PR[91,2] = PR[90,2] + 13.339;
   1:  PR[91,3] = PR[90,3] + 62.079;
   1:L PR[91] R[100]mm/sec CNT100;
   1:  PR[91,1] = PR[90,1] + 70.861;
   1:  PR[91,2] = PR[90,2] + 17.306;
   1:  PR[91,3] = PR[90,3] + 62.098;
   1:L PR[91] R[100]mm/sec CNT100;
   1:  PR[91,1] = PR[90,1] + 65.259;
   1:  PR[91,2] = PR[90,2] + 20.588;
   1:  PR[91,3] = PR[90,3] + 62.118;
   1:L PR[91] R[100]mm/sec CNT100;
   1:  PR[91,1] = PR[90,1] + 62.348;
   1:  PR[91,2] = PR[90,2] + 21.624;
   1:  PR[91,3] = PR[90,3] + 62.141;
   1:L PR[91] R[100]mm/sec CNT100;
   1:  PR[91,1] = PR[90,1] + 58.554;
   1:  PR[91,2] = PR[90,2] + 22.860;
   1:  PR[91,3] = PR[90,3] + 62.151;
   1:L PR[91] R[100]mm/sec CNT100;
   1:  PR[91,1] = PR[90,1] + 55.841;
   1:  PR[91,2] = PR[90,2] + 23.361;
   1:  PR[91,3] = PR[90,3] + 62.165;
   1:L PR[91] R[100]mm/sec CNT100;
   1:  PR[91,1] = PR[90,1] + 52.622;
   1:  PR[91,2] = PR[90,2] + 23.872;
   1:  PR[91,3] = PR[90,3] + 62.175;
   1:L PR[91] R[100]mm/sec CNT100;
   1:  PR[91,1] = PR[90,1] + 49.696;
   1:  PR[91,2] = PR[90,2] + 24.043;
   1:  PR[91,3] = PR[90,3] + 62.186;
   1:L PR[91] R[100]mm/sec CNT100;
   1:  PR[91,1] = PR[90,1] + 47.890;
   1:  PR[91,2] = PR[90,2] + 24.173;
   1:  PR[91,3] = PR[90,3] + 62.196;
   1:L PR[91] R[100]mm/sec CNT100;
   1:  PR[91,1] = PR[90,1] + 43.942;
   1:  PR[91,2] = PR[90,2] + 24.100;
   1:  PR[91,3] = PR[90,3] + 62.202;
   1:L PR[91] R[100]mm/sec CNT100;
   1:  PR[91,1] = PR[90,1] + 43.559;
   1:  PR[91,2] = PR[90,2] + 24.084;
   1:  PR[91,3] = PR[90,3] + 62.216;
   1:L PR[91] R[100]mm/sec CNT100;
   1:  PR[91,1] = PR[90,1] + 37.882;
   1:  PR[91,2] = PR[90,2] + 23.348;
   1:  PR[91,3] = PR[90,3] + 62.217;
   1:L PR[91] R[100]mm/sec CNT100;
   1:  PR[91,1] = PR[90,1] + 31.882;
   1:  PR[91,2] = PR[90,2] + 21.740;
   1:  PR[91,3] = PR[90,3] + 62.237;
   1:L PR[91] R[100]mm/sec CNT100;
   1:  PR[91,1] = PR[90,1] + 30.835;
   1:  PR[91,2] = PR[90,2] + 21.417;
   1:  PR[91,3] = PR[90,3] + 62.258;
   1:L PR[91] R[100]mm/sec CNT100;
   1:  PR[91,1] = PR[90,1] + 29.883;
   1:  PR[91,2] = PR[90,2] + 21.785;
   1:  PR[91,3] = PR[90,3] + 62.262;
   1:L PR[91] R[100]mm/sec CNT100;
   1:  PR[91,1] = PR[90,1] + 28.886;
   1:  PR[91,2] = PR[90,2] + 22.112;
   1:  PR[91,3] = PR[90,3] + 62.265;
   1:L PR[91] R[100]mm/sec CNT100;
   1:  PR[91,1] = PR[90,1] + 27.266;
   1:  PR[91,2] = PR[90,2] + 22.428;
   1:  PR[91,3] = PR[90,3] + 62.269;
   1:L PR[91] R[100]mm/sec CNT100;
   1:  PR[91,1] = PR[90,1] + 26.958;
   1:  PR[91,2] = PR[90,2] + 22.501;
   1:  PR[91,3] = PR[90,3] + 62.274;
   1:L PR[91] R[100]mm/sec CNT100;
   1:  PR[91,1] = PR[90,1] + 23.155;
   1:  PR[91,2] = PR[90,2] + 23.213;
   1:  PR[91,3] = PR[90,3] + 62.275;
   1:L PR[91] R[100]mm/sec CNT100;
   1:  PR[91,1] = PR[90,1] + 18.846;
   1:  PR[91,2] = PR[90,2] + 23.041;
   1:  PR[91,3] = PR[90,3] + 62.289;
   1:L PR[91] R[100]mm/sec CNT100;
   1:  PR[91,1] = PR[90,1] + 17.568;
   1:  PR[91,2] = PR[90,2] + 22.971;
   1:  PR[91,3] = PR[90,3] + 62.304;
   1:L PR[91] R[100]mm/sec CNT100;
   1:  PR[91,1] = PR[90,1] + 13.157;
   1:  PR[91,2] = PR[90,2] + 21.768;
   1:  PR[91,3] = PR[90,3] + 62.308;
   1:L PR[91] R[100]mm/sec CNT100;
   1:  PR[91,1] = PR[90,1] + 12.218;
   1:  PR[91,2] = PR[90,2] + 21.475;
   1:  PR[91,3] = PR[90,3] + 62.324;
   1:L PR[91] R[100]mm/sec CNT100;
   1:  PR[91,1] = PR[90,1] + 7.861;
   1:  PR[91,2] = PR[90,2] + 19.112;
   1:  PR[91,3] = PR[90,3] + 62.327;
   1:L PR[91] R[100]mm/sec CNT100;
   1:  PR[91,1] = PR[90,1] + 7.310;
   1:  PR[91,2] = PR[90,2] + 18.772;
   1:  PR[91,3] = PR[90,3] + 62.344;
   1:L PR[91] R[100]mm/sec CNT100;
   1:  PR[91,1] = PR[90,1] + 5.820;
   1:  PR[91,2] = PR[90,2] + 17.542;
   1:  PR[91,3] = PR[90,3] + 62.346;
   1:L PR[91] R[100]mm/sec CNT100;
   1:  PR[91,1] = PR[90,1] + 2.584;
   1:  PR[91,2] = PR[90,2] + 19.244;
   1:  PR[91,3] = PR[90,3] + 62.353;
   1:L PR[91] R[100]mm/sec CNT100;
   1:  PR[91,1] = PR[90,1] + 1.526;
   1:  PR[91,2] = PR[90,2] + 19.758;
   1:  PR[91,3] = PR[90,3] + 62.365;
   1:L PR[91] R[100]mm/sec CNT100;
   1:  PR[91,1] = PR[90,1] + -3.316;
   1:  PR[91,2] = PR[90,2] + 21.198;
   1:  PR[91,3] = PR[90,3] + 62.369;
   1:L PR[91] R[100]mm/sec CNT100;
   1:  PR[91,1] = PR[90,1] + -4.137;
   1:  PR[91,2] = PR[90,2] + 21.465;
   1:  PR[91,3] = PR[90,3] + 62.387;
   1:L PR[91] R[100]mm/sec CNT100;
   1:  PR[91,1] = PR[90,1] + -9.732;
   1:  PR[91,2] = PR[90,2] + 22.117;
   1:  PR[91,3] = PR[90,3] + 62.390;
   1:L PR[91] R[100]mm/sec CNT100;
   1:  PR[91,1] = PR[90,1] + -15.414;
   1:  PR[91,2] = PR[90,2] + 21.677;
   1:  PR[91,3] = PR[90,3] + 62.409;
   1:L PR[91] R[100]mm/sec CNT100;
   1:  PR[91,1] = PR[90,1] + -17.544;
   1:  PR[91,2] = PR[90,2] + 21.110;
   1:  PR[91,3] = PR[90,3] + 62.429;
   1:L PR[91] R[100]mm/sec CNT100;
   1:  PR[91,1] = PR[90,1] + -20.834;
   1:  PR[91,2] = PR[90,2] + 20.156;
   1:  PR[91,3] = PR[90,3] + 62.436;
   1:L PR[91] R[100]mm/sec CNT100;
   1:  PR[91,1] = PR[90,1] + -22.439;
   1:  PR[91,2] = PR[90,2] + 19.468;
   1:  PR[91,3] = PR[90,3] + 62.448;
   1:L PR[91] R[100]mm/sec CNT100;
   1:  PR[91,1] = PR[90,1] + -25.687;
   1:  PR[91,2] = PR[90,2] + 17.708;
   1:  PR[91,3] = PR[90,3] + 62.454;
   1:L PR[91] R[100]mm/sec CNT100;
   1:  PR[91,1] = PR[90,1] + -30.477;
   1:  PR[91,2] = PR[90,2] + 18.910;
   1:  PR[91,3] = PR[90,3] + 62.467;
   1:L PR[91] R[100]mm/sec CNT100;
   1:  PR[91,1] = PR[90,1] + -32.485;
   1:  PR[91,2] = PR[90,2] + 19.608;
   1:  PR[91,3] = PR[90,3] + 62.484;
   1:L PR[91] R[100]mm/sec CNT100;
   1:  PR[91,1] = PR[90,1] + -36.962;
   1:  PR[91,2] = PR[90,2] + 20.623;
   1:  PR[91,3] = PR[90,3] + 62.491;
   1:L PR[91] R[100]mm/sec CNT100;
   1:  PR[91,1] = PR[90,1] + -38.494;
   1:  PR[91,2] = PR[90,2] + 20.913;
   1:  PR[91,3] = PR[90,3] + 62.507;
   1:L PR[91] R[100]mm/sec CNT100;
   1:  PR[91,1] = PR[90,1] + -39.263;
   1:  PR[91,2] = PR[90,2] + 20.978;
   1:  PR[91,3] = PR[90,3] + 62.512;
   1:L PR[91] R[100]mm/sec CNT100;
   1:  PR[91,1] = PR[90,1] + -43.956;
   1:  PR[91,2] = PR[90,2] + 21.605;
   1:  PR[91,3] = PR[90,3] + 62.515;
   1:L PR[91] R[100]mm/sec CNT100;
   1:  PR[91,1] = PR[90,1] + -48.315;
   1:  PR[91,2] = PR[90,2] + 21.945;
   1:  PR[91,3] = PR[90,3] + 62.531;
   1:L PR[91] R[100]mm/sec CNT100;
   1:  PR[91,1] = PR[90,1] + -49.009;
   1:  PR[91,2] = PR[90,2] + 21.934;
   1:  PR[91,3] = PR[90,3] + 62.546;
   1:L PR[91] R[100]mm/sec CNT100;
   1:  PR[91,1] = PR[90,1] + -53.804;
   1:  PR[91,2] = PR[90,2] + 21.680;
   1:  PR[91,3] = PR[90,3] + 62.548;
   1:L PR[91] R[100]mm/sec CNT100;
   1:  PR[91,1] = PR[90,1] + -55.903;
   1:  PR[91,2] = PR[90,2] + 21.548;
   1:  PR[91,3] = PR[90,3] + 62.565;
   1:L PR[91] R[100]mm/sec CNT100;
   1:  PR[91,1] = PR[90,1] + -58.203;
   1:  PR[91,2] = PR[90,2] + 21.060;
   1:  PR[91,3] = PR[90,3] + 62.572;
   1:L PR[91] R[100]mm/sec CNT100;
   1:  PR[91,1] = PR[90,1] + -62.476;
   1:  PR[91,2] = PR[90,2] + 20.112;
   1:  PR[91,3] = PR[90,3] + 62.580;
   1:L PR[91] R[100]mm/sec CNT100;
   1:  PR[91] = PR[90];
   1:  PR[91,1] = PR[90,1] + -64.703;
   1:  PR[91,2] = PR[90,2] + 18.964;
   1:  PR[91,3] = PR[90,3] + 63.895;
   1:L PR[91] R[100]mm/sec CNT100;
   1:  PR[91,1] = PR[90,1] + -66.880;
   1:  PR[91,2] = PR[90,2] + 18.036;
   1:  PR[91,3] = PR[90,3] + 62.608;
   1:L PR[91] R[100]mm/sec CNT100;
   1:  PR[91,1] = PR[90,1] + -69.959;
   1:  PR[91,2] = PR[90,2] + 16.004;
   1:  PR[91,3] = PR[90,3] + 62.616;
   1:L PR[91] R[100]mm/sec CNT100;
   1:  PR[91,1] = PR[90,1] + -71.348;
   1:  PR[91,2] = PR[90,2] + 15.072;
   1:  PR[91,3] = PR[90,3] + 62.629;
   1:L PR[91] R[100]mm/sec CNT100;
   1:  PR[91,1] = PR[90,1] + -74.886;
   1:  PR[91,2] = PR[90,2] + 11.557;
   1:  PR[91,3] = PR[90,3] + 62.634;
   1:L PR[91] R[100]mm/sec CNT100;
   1:  PR[91,1] = PR[90,1] + -77.433;
   1:  PR[91,2] = PR[90,2] + 7.661;
   1:  PR[91,3] = PR[90,3] + 62.652;
   1:L PR[91] R[100]mm/sec CNT100;
   1:  PR[91,1] = PR[90,1] + -78.963;
   1:  PR[91,2] = PR[90,2] + 3.522;
   1:  PR[91,3] = PR[90,3] + 62.668;
   1:L PR[91] R[100]mm/sec CNT100;
   1:  PR[91,1] = PR[90,1] + -79.436;
   1:  PR[91,2] = PR[90,2] + -0.397;
   1:  PR[91,3] = PR[90,3] + 62.683;
   1:L PR[91] R[100]mm/sec CNT100;
   1:  PR[91,1] = PR[90,1] + -79.491;
   1:  PR[91,2] = PR[90,2] + -0.700;
   1:  PR[91,3] = PR[90,3] + 62.697;
   1:L PR[91] R[100]mm/sec CNT100;
   1:  PR[91,1] = PR[90,1] + -79.190;
   1:  PR[91,2] = PR[90,2] + -2.135;
   1:  PR[91,3] = PR[90,3] + 62.698;
   1:L PR[91] R[100]mm/sec CNT100;
   1:  PR[91,1] = PR[90,1] + -78.822;
   1:  PR[91,2] = PR[90,2] + -5.152;
   1:  PR[91,3] = PR[90,3] + 62.703;
   1:L PR[91] R[100]mm/sec CNT100;
   1:  PR[91,1] = PR[90,1] + -78.366;
   1:  PR[91,2] = PR[90,2] + -6.421;
   1:  PR[91,3] = PR[90,3] + 62.714;
   1:L PR[91] R[100]mm/sec CNT100;
   1:  PR[91,1] = PR[90,1] + -77.219;
   1:  PR[91,2] = PR[90,2] + -9.458;
   1:  PR[91,3] = PR[90,3] + 62.718;
   1:L PR[91] R[100]mm/sec CNT100;
   1:  PR[91,1] = PR[90,1] + -76.679;
   1:  PR[91,2] = PR[90,2] + -10.309;
   1:  PR[91,3] = PR[90,3] + 62.729;
   1:L PR[91] R[100]mm/sec CNT100;
   1:  PR[91,1] = PR[90,1] + -74.520;
   1:  PR[91,2] = PR[90,2] + -13.521;
   1:  PR[91,3] = PR[90,3] + 62.733;
   1:L PR[91] R[100]mm/sec CNT100;
   1:  PR[91,1] = PR[90,1] + -74.220;
   1:  PR[91,2] = PR[90,2] + -13.829;
   1:  PR[91,3] = PR[90,3] + 62.746;
   1:L PR[91] R[100]mm/sec CNT100;
   1:  PR[91,1] = PR[90,1] + -71.709;
   1:  PR[91,2] = PR[90,2] + -16.223;
   1:  PR[91,3] = PR[90,3] + 62.748;
   1:L PR[91] R[100]mm/sec CNT100;
   1:  PR[91,1] = PR[90,1] + -70.749;
   1:  PR[91,2] = PR[90,2] + -17.079;
   1:  PR[91,3] = PR[90,3] + 62.760;
   1:L PR[91] R[100]mm/sec CNT100;
   1:  PR[91,1] = PR[90,1] + -65.793;
   1:  PR[91,2] = PR[90,2] + -19.997;
   1:  PR[91,3] = PR[90,3] + 62.764;
   1:L PR[91] R[100]mm/sec CNT100;
   1:  PR[91,1] = PR[90,1] + -62.716;
   1:  PR[91,2] = PR[90,2] + -21.151;
   1:  PR[91,3] = PR[90,3] + 62.784;
   1:L PR[91] R[100]mm/sec CNT100;
   1:  PR[91,1] = PR[90,1] + -60.061;
   1:  PR[91,2] = PR[90,2] + -22.120;
   1:  PR[91,3] = PR[90,3] + 62.796;
   1:L PR[91] R[100]mm/sec CNT100;
   1:  PR[91,1] = PR[90,1] + -53.804;
   1:  PR[91,2] = PR[90,2] + -23.312;
   1:  PR[91,3] = PR[90,3] + 62.805;
   1:L PR[91] R[100]mm/sec CNT100;
   1:  PR[91,1] = PR[90,1] + -52.790;
   1:  PR[91,2] = PR[90,2] + -23.410;
   1:  PR[91,3] = PR[90,3] + 62.827;
   1:L PR[91] R[100]mm/sec CNT100;
   1:  PR[91,1] = PR[90,1] + -47.969;
   1:  PR[91,2] = PR[90,2] + -23.606;
   1:  PR[91,3] = PR[90,3] + 62.831;
   1:L PR[91] R[100]mm/sec CNT100;
   1:  PR[91,1] = PR[90,1] + -42.146;
   1:  PR[91,2] = PR[90,2] + -23.350;
   1:  PR[91,3] = PR[90,3] + 62.848;
   1:L PR[91] R[100]mm/sec CNT100;
   1:  PR[91,1] = PR[90,1] + -36.916;
   1:  PR[91,2] = PR[90,2] + -22.620;
   1:  PR[91,3] = PR[90,3] + 62.868;
   1:L PR[91] R[100]mm/sec CNT100;
   1:  PR[91,1] = PR[90,1] + -32.017;
   1:  PR[91,2] = PR[90,2] + -21.654;
   1:  PR[91,3] = PR[90,3] + 62.886;
   1:L PR[91] R[100]mm/sec CNT100;
   1:  PR[91,1] = PR[90,1] + -31.063;
   1:  PR[91,2] = PR[90,2] + -21.524;
   1:  PR[91,3] = PR[90,3] + 62.903;
   1:L PR[91] R[100]mm/sec CNT100;
   1:  PR[91,1] = PR[90,1] + -29.599;
   1:  PR[91,2] = PR[90,2] + -21.187;
   1:  PR[91,3] = PR[90,3] + 62.907;
   1:L PR[91] R[100]mm/sec CNT100;
   1:  PR[91,1] = PR[90,1] + -24.376;
   1:  PR[91,2] = PR[90,2] + -19.798;
   1:  PR[91,3] = PR[90,3] + 62.912;
   1:L PR[91] R[100]mm/sec CNT100;
   1:  PR[91,1] = PR[90,1] + -22.419;
   1:  PR[91,2] = PR[90,2] + -20.865;
   1:  PR[91,3] = PR[90,3] + 62.931;
   1:L PR[91] R[100]mm/sec CNT100;
   1:  PR[91,1] = PR[90,1] + -20.179;
   1:  PR[91,2] = PR[90,2] + -21.826;
   1:  PR[91,3] = PR[90,3] + 62.938;
   1:L PR[91] R[100]mm/sec CNT100;
   1:  PR[91,1] = PR[90,1] + -17.442;
   1:  PR[91,2] = PR[90,2] + -22.624;
   1:  PR[91,3] = PR[90,3] + 62.947;
   1:L PR[91] R[100]mm/sec CNT100;
   1:  PR[91,1] = PR[90,1] + -14.775;
   1:  PR[91,2] = PR[90,2] + -23.334;
   1:  PR[91,3] = PR[90,3] + 62.957;
   1:L PR[91] R[100]mm/sec CNT100;
   1:  PR[91,1] = PR[90,1] + -9.081;
   1:  PR[91,2] = PR[90,2] + -23.778;
   1:  PR[91,3] = PR[90,3] + 62.966;
   1:L PR[91] R[100]mm/sec CNT100;
   1:  PR[91,1] = PR[90,1] + -5.385;
   1:  PR[91,2] = PR[90,2] + -23.350;
   1:  PR[91,3] = PR[90,3] + 62.986;
   1:L PR[91] R[100]mm/sec CNT100;
   1:  PR[91,1] = PR[90,1] + -3.330;
   1:  PR[91,2] = PR[90,2] + -23.143;
   1:  PR[91,3] = PR[90,3] + 62.999;
   1:L PR[91] R[100]mm/sec CNT100;
   1:  PR[91,1] = PR[90,1] + 2.423;
   1:  PR[91,2] = PR[90,2] + -21.444;
   1:  PR[91,3] = PR[90,3] + 63.006;
   1:L PR[91] R[100]mm/sec CNT100;
   1:  PR[91,1] = PR[90,1] + 4.280;
   1:  PR[91,2] = PR[90,2] + -20.543;
   1:  PR[91,3] = PR[90,3] + 63.027;
   1:L PR[91] R[100]mm/sec CNT100;
   1:  PR[91,1] = PR[90,1] + 6.054;
   1:  PR[91,2] = PR[90,2] + -19.623;
   1:  PR[91,3] = PR[90,3] + 63.034;
   1:L PR[91] R[100]mm/sec CNT100;
   1:  PR[91,1] = PR[90,1] + 7.161;
   1:  PR[91,2] = PR[90,2] + -20.491;
   1:  PR[91,3] = PR[90,3] + 63.041;
   1:L PR[91] R[100]mm/sec CNT100;
   1:  PR[91,1] = PR[90,1] + 7.243;
   1:  PR[91,2] = PR[90,2] + -20.542;
   1:  PR[91,3] = PR[90,3] + 63.046;
   1:L PR[91] R[100]mm/sec CNT100;
   1:  PR[91,1] = PR[90,1] + 12.095;
   1:  PR[91,2] = PR[90,2] + -23.169;
   1:L PR[91] R[100]mm/sec CNT100;
   1:  PR[91,1] = PR[90,1] + 12.482;
   1:  PR[91,2] = PR[90,2] + -23.290;
   1:  PR[91,3] = PR[90,3] + 63.065;
   1:L PR[91] R[100]mm/sec CNT100;
   1:  PR[91,1] = PR[90,1] + 17.448;
   1:  PR[91,2] = PR[90,2] + -24.643;
   1:  PR[91,3] = PR[90,3] + 63.067;
   1:L PR[91] R[100]mm/sec CNT100;
   1:  PR[91,1] = PR[90,1] + 18.152;
   1:  PR[91,2] = PR[90,2] + -24.682;
   1:  PR[91,3] = PR[90,3] + 63.085;
   1:L PR[91] R[100]mm/sec CNT100;
   1:  PR[91,1] = PR[90,1] + 23.030;
   1:  PR[91,2] = PR[90,2] + -24.877;
   1:  PR[91,3] = PR[90,3] + 63.087;
   1:L PR[91] R[100]mm/sec CNT100;
   1:  PR[91,1] = PR[90,1] + 28.628;
   1:  PR[91,2] = PR[90,2] + -23.818;
   1:  PR[91,3] = PR[90,3] + 63.104;
   1:L PR[91] R[100]mm/sec CNT100;
   1:  PR[91,1] = PR[90,1] + 30.272;
   1:  PR[91,2] = PR[90,2] + -23.289;
   1:  PR[91,3] = PR[90,3] + 63.124;
   1:L PR[91] R[100]mm/sec CNT100;
   1:  PR[91,1] = PR[90,1] + 31.868;
   1:  PR[91,2] = PR[90,2] + -23.743;
   1:  PR[91,3] = PR[90,3] + 63.130;
   1:L PR[91] R[100]mm/sec CNT100;
   1:  PR[91,1] = PR[90,1] + 36.595;
   1:  PR[91,2] = PR[90,2] + -25.013;
   1:  PR[91,3] = PR[90,3] + 63.135;
   1:L PR[91] R[100]mm/sec CNT100;
   1:  PR[91,1] = PR[90,1] + 42.457;
   1:  PR[91,2] = PR[90,2] + -25.767;
   1:  PR[91,3] = PR[90,3] + 63.152;
   1:L PR[91] R[100]mm/sec CNT100;
   1:  PR[91,1] = PR[90,1] + 44.380;
   1:  PR[91,2] = PR[90,2] + -25.774;
   1:  PR[91,3] = PR[90,3] + 63.173;
   1:L PR[91] R[100]mm/sec CNT100;
   1:  PR[91,1] = PR[90,1] + 47.255;
   1:  PR[91,2] = PR[90,2] + -25.827;
   1:  PR[91,3] = PR[90,3] + 63.180;
   1:L PR[91] R[100]mm/sec CNT100;
   1:  PR[91,1] = PR[90,1] + 50.892;
   1:  PR[91,2] = PR[90,2] + -25.566;
   1:  PR[91,3] = PR[90,3] + 63.189;
   1:L PR[91] R[100]mm/sec CNT100;
   1:  PR[91,1] = PR[90,1] + 51.866;
   1:  PR[91,2] = PR[90,2] + -25.509;
   1:  PR[91,3] = PR[90,3] + 63.202;
   1:L PR[91] R[100]mm/sec CNT100;
   1:  PR[91,1] = PR[90,1] + 52.917;
   1:  PR[91,2] = PR[90,2] + -25.343;
   1:  PR[91,3] = PR[90,3] + 63.205;
   1:L PR[91] R[100]mm/sec CNT100;
   1:  PR[91,1] = PR[90,1] + 57.484;
   1:  PR[91,2] = PR[90,2] + -24.500;
   1:  PR[91,3] = PR[90,3] + 63.209;
   1:L PR[91] R[100]mm/sec CNT100;
